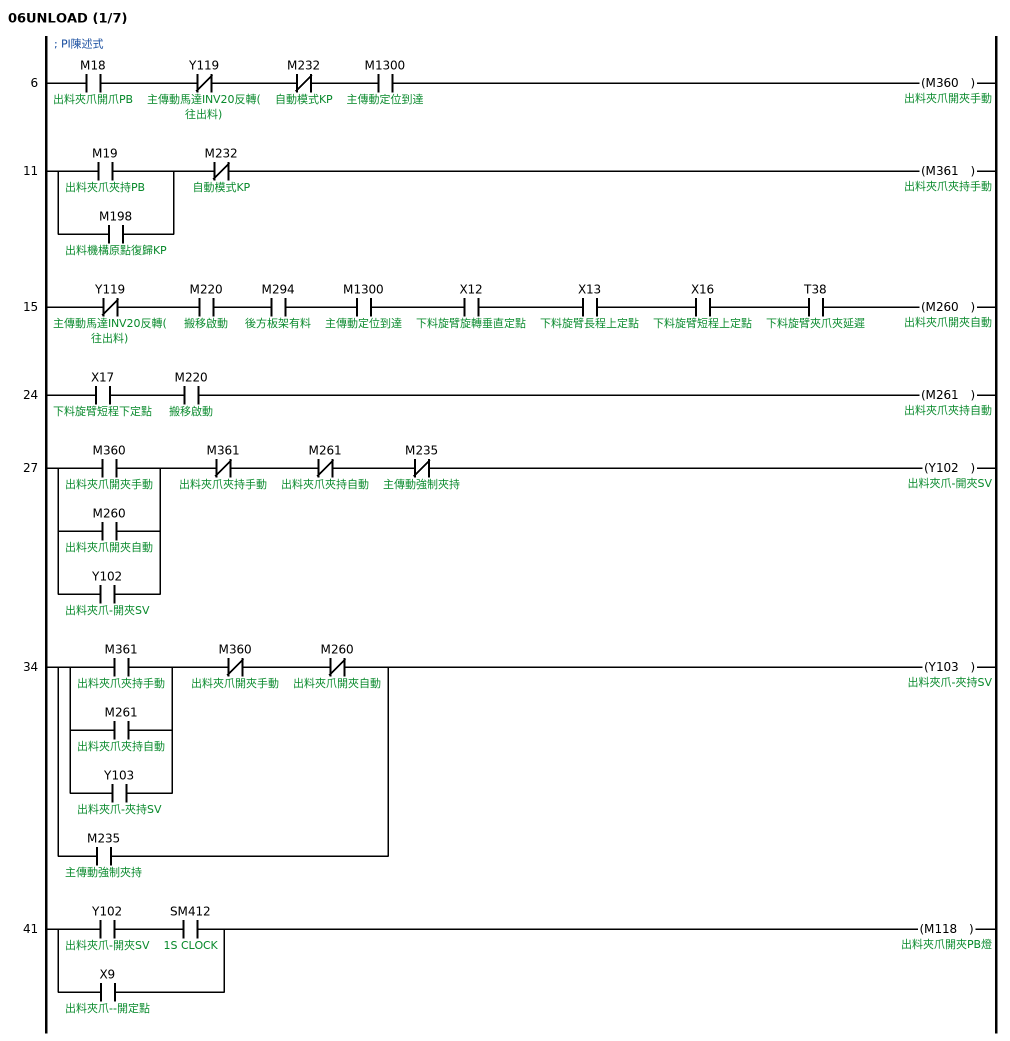
[picture p24: ladder of 06UNLOAD, rungs at steps 6 to 41]
; PI陳述式
6     LD      M18  ; 出料夾爪開爪PB
      ANI     Y119  ; 主傳動馬達INV20反轉(往出料)
      ANI     M232  ; 自動模式KP
      AND     M1300  ; 主傳動定位到達
      OUT     M360  ; 出料夾爪開夾手動
11    LD      M19  ; 出料夾爪夾持PB
      OR      M198  ; 出料機構原點復歸KP
      ANI     M232  ; 自動模式KP
      OUT     M361  ; 出料夾爪夾持手動
15    LDI     Y119  ; 主傳動馬達INV20反轉(往出料)
      AND     M220  ; 搬移啟動
      AND     M294  ; 後方板架有料
      AND     M1300  ; 主傳動定位到達
      AND     X12  ; 下料旋臂旋轉垂直定點
      AND     X13  ; 下料旋臂長程上定點
      AND     X16  ; 下料旋臂短程上定點
      AND     T38  ; 下料旋臂夾爪夾延遲
      OUT     M260  ; 出料夾爪開夾自動
24    LD      X17  ; 下料旋臂短程下定點
      AND     M220  ; 搬移啟動
      OUT     M261  ; 出料夾爪夾持自動
27    LD      M360  ; 出料夾爪開夾手動
      OR      M260  ; 出料夾爪開夾自動
      OR      Y102  ; 出料夾爪-開夾SV
      ANI     M361  ; 出料夾爪夾持手動
      ANI     M261  ; 出料夾爪夾持自動
      ANI     M235  ; 主傳動強制夾持
      OUT     Y102  ; 出料夾爪-開夾SV
34    LD      M361  ; 出料夾爪夾持手動
      OR      M261  ; 出料夾爪夾持自動
      OR      Y103  ; 出料夾爪-夾持SV
      ANI     M360  ; 出料夾爪開夾手動
      ANI     M260  ; 出料夾爪開夾自動
      OR      M235  ; 主傳動強制夾持
      OUT     Y103  ; 出料夾爪-夾持SV
41    LD      Y102  ; 出料夾爪-開夾SV
      AND     SM412  ; 1S CLOCK
      OR      X9  ; 出料夾爪--開定點
      OUT     M118  ; 出料夾爪開夾PB燈
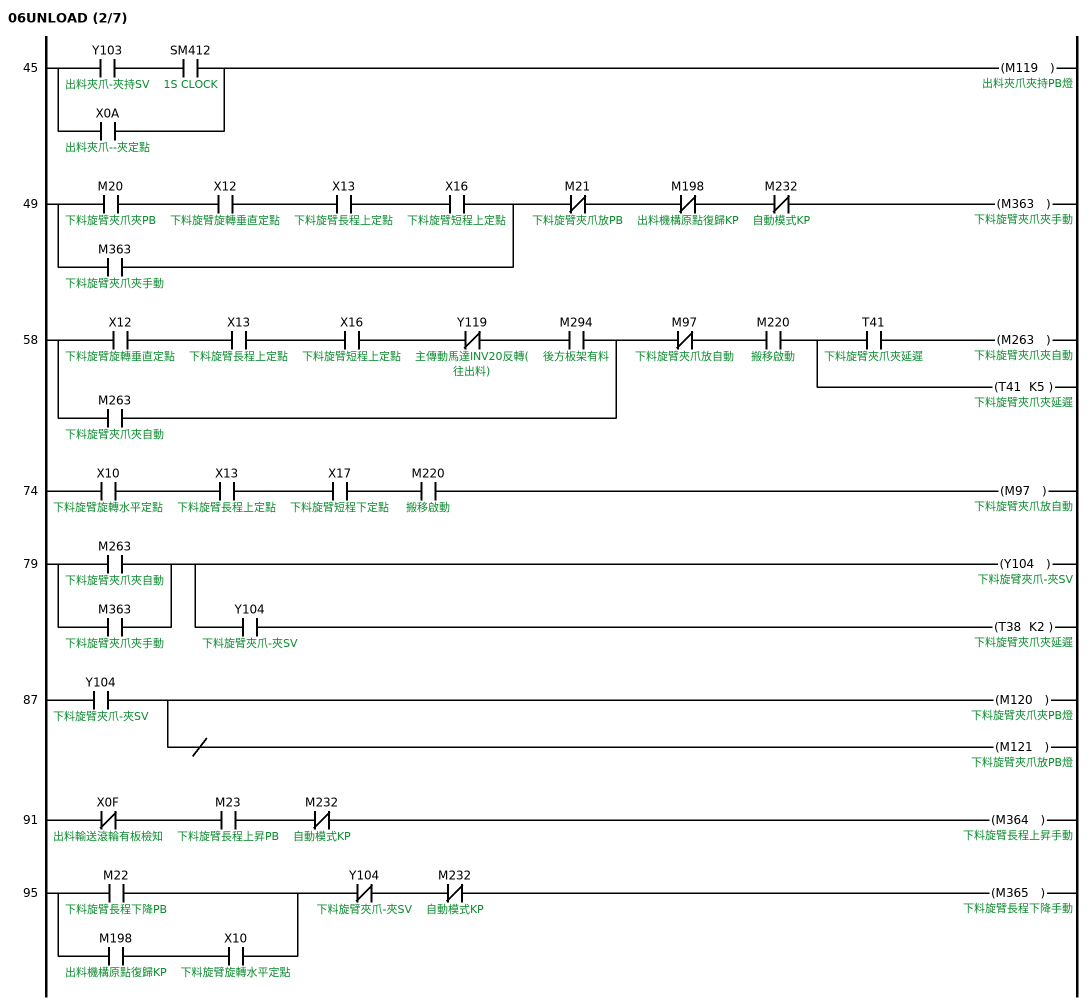
45    LD      Y103  ; 出料夾爪-夾持SV
      AND     SM412  ; 1S CLOCK
      OR      X0A  ; 出料夾爪--夾定點
      OUT     M119  ; 出料夾爪夾持PB燈
49    LD      M20  ; 下料旋臂夾爪夾PB
      AND     X12  ; 下料旋臂旋轉垂直定點
      AND     X13  ; 下料旋臂長程上定點
      AND     X16  ; 下料旋臂短程上定點
      OR      M363  ; 下料旋臂夾爪夾手動
      ANI     M21  ; 下料旋臂夾爪放PB
      ANI     M198  ; 出料機構原點復歸KP
      ANI     M232  ; 自動模式KP
      OUT     M363  ; 下料旋臂夾爪夾手動
58    LD      X12  ; 下料旋臂旋轉垂直定點
      AND     X13  ; 下料旋臂長程上定點
      AND     X16  ; 下料旋臂短程上定點
      ANI     Y119  ; 主傳動馬達INV20反轉(往出料)
      AND     M294  ; 後方板架有料
      OR      M263  ; 下料旋臂夾爪夾自動
      ANI     M97  ; 下料旋臂夾爪放自動
      AND     M220  ; 搬移啟動
      MPS
      AND     T41  ; 下料旋臂夾爪夾延遲
      OUT     M263  ; 下料旋臂夾爪夾自動
      MPP
      OUT     T41 K5  ; 下料旋臂夾爪夾延遲
74    LD      X10  ; 下料旋臂旋轉水平定點
      AND     X13  ; 下料旋臂長程上定點
      AND     X17  ; 下料旋臂短程下定點
      AND     M220  ; 搬移啟動
      OUT     M97  ; 下料旋臂夾爪放自動
79    LD      M263  ; 下料旋臂夾爪夾自動
      OR      M363  ; 下料旋臂夾爪夾手動
      OUT     Y104  ; 下料旋臂夾爪-夾SV
      AND     Y104  ; 下料旋臂夾爪-夾SV
      OUT     T38 K2  ; 下料旋臂夾爪夾延遲
87    LD      Y104  ; 下料旋臂夾爪-夾SV
      OUT     M120  ; 下料旋臂夾爪夾PB燈
      INV
      OUT     M121  ; 下料旋臂夾爪放PB燈
91    LDI     X0F  ; 出料輸送滾輪有板檢知
      AND     M23  ; 下料旋臂長程上昇PB
      ANI     M232  ; 自動模式KP
      OUT     M364  ; 下料旋臂長程上昇手動
95    LD      M22  ; 下料旋臂長程下降PB
      LD      M198  ; 出料機構原點復歸KP
      AND     X10  ; 下料旋臂旋轉水平定點
      ORB
      ANI     Y104  ; 下料旋臂夾爪-夾SV
      ANI     M232  ; 自動模式KP
      OUT     M365  ; 下料旋臂長程下降手動
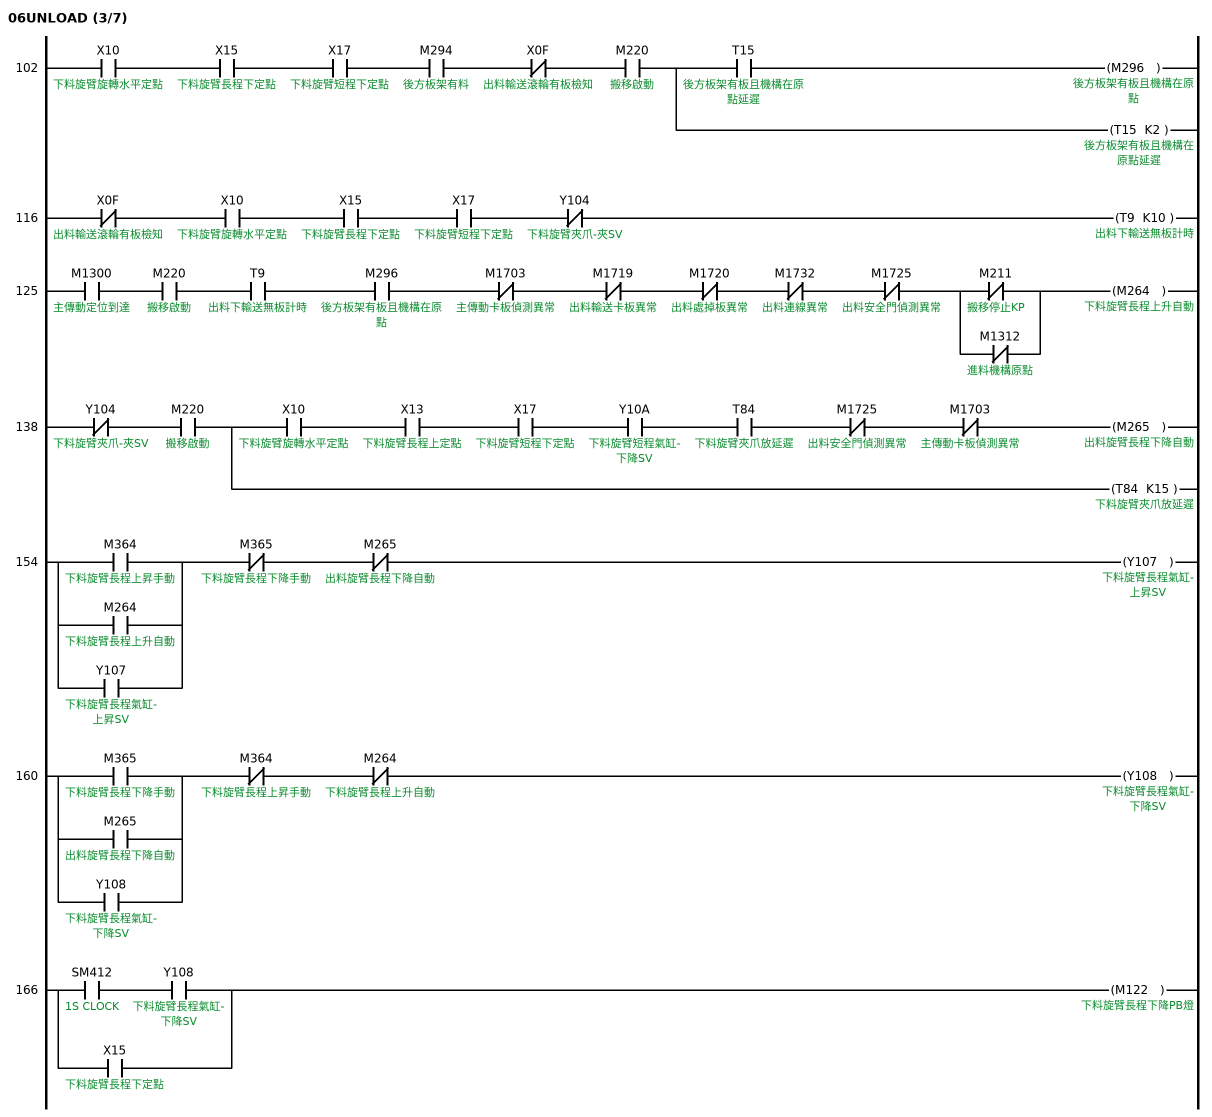
102   LD      X10  ; 下料旋臂旋轉水平定點
      AND     X15  ; 下料旋臂長程下定點
      AND     X17  ; 下料旋臂短程下定點
      AND     M294  ; 後方板架有料
      ANI     X0F  ; 出料輸送滾輪有板檢知
      AND     M220  ; 搬移啟動
      MPS
      AND     T15  ; 後方板架有板且機構在原點延遲
      OUT     M296  ; 後方板架有板且機構在原點
      MPP
      OUT     T15 K2  ; 後方板架有板且機構在原點延遲
116   LDI     X0F  ; 出料輸送滾輪有板檢知
      AND     X10  ; 下料旋臂旋轉水平定點
      AND     X15  ; 下料旋臂長程下定點
      AND     X17  ; 下料旋臂短程下定點
      ANI     Y104  ; 下料旋臂夾爪-夾SV
      OUT     T9 K10  ; 出料下輸送無板計時
125   LD      M1300  ; 主傳動定位到達
      AND     M220  ; 搬移啟動
      AND     T9  ; 出料下輸送無板計時
      AND     M296  ; 後方板架有板且機構在原點
      ANI     M1703  ; 主傳動卡板偵測異常
      ANI     M1719  ; 出料輸送卡板異常
      ANI     M1720  ; 出料處掉板異常
      ANI     M1732  ; 出料連線異常
      ANI     M1725  ; 出料安全門偵測異常
      LDI     M211  ; 搬移停止KP
      ORI     M1312  ; 進料機構原點
      ANB
      OUT     M264  ; 下料旋臂長程上升自動
138   LDI     Y104  ; 下料旋臂夾爪-夾SV
      AND     M220  ; 搬移啟動
      MPS
      AND     X10  ; 下料旋臂旋轉水平定點
      AND     X13  ; 下料旋臂長程上定點
      AND     X17  ; 下料旋臂短程下定點
      AND     Y10A  ; 下料旋臂短程氣缸-下降SV
      AND     T84  ; 下料旋臂夾爪放延遲
      ANI     M1725  ; 出料安全門偵測異常
      ANI     M1703  ; 主傳動卡板偵測異常
      OUT     M265  ; 出料旋臂長程下降自動
      MPP
      OUT     T84 K15  ; 下料旋臂夾爪放延遲
154   LD      M364  ; 下料旋臂長程上昇手動
      OR      M264  ; 下料旋臂長程上升自動
      OR      Y107  ; 下料旋臂長程氣缸-上昇SV
      ANI     M365  ; 下料旋臂長程下降手動
      ANI     M265  ; 出料旋臂長程下降自動
      OUT     Y107  ; 下料旋臂長程氣缸-上昇SV
160   LD      M365  ; 下料旋臂長程下降手動
      OR      M265  ; 出料旋臂長程下降自動
      OR      Y108  ; 下料旋臂長程氣缸-下降SV
      ANI     M364  ; 下料旋臂長程上昇手動
      ANI     M264  ; 下料旋臂長程上升自動
      OUT     Y108  ; 下料旋臂長程氣缸-下降SV
166   LD      SM412  ; 1S CLOCK
      AND     Y108  ; 下料旋臂長程氣缸-下降SV
      OR      X15  ; 下料旋臂長程下定點
      OUT     M122  ; 下料旋臂長程下降PB燈
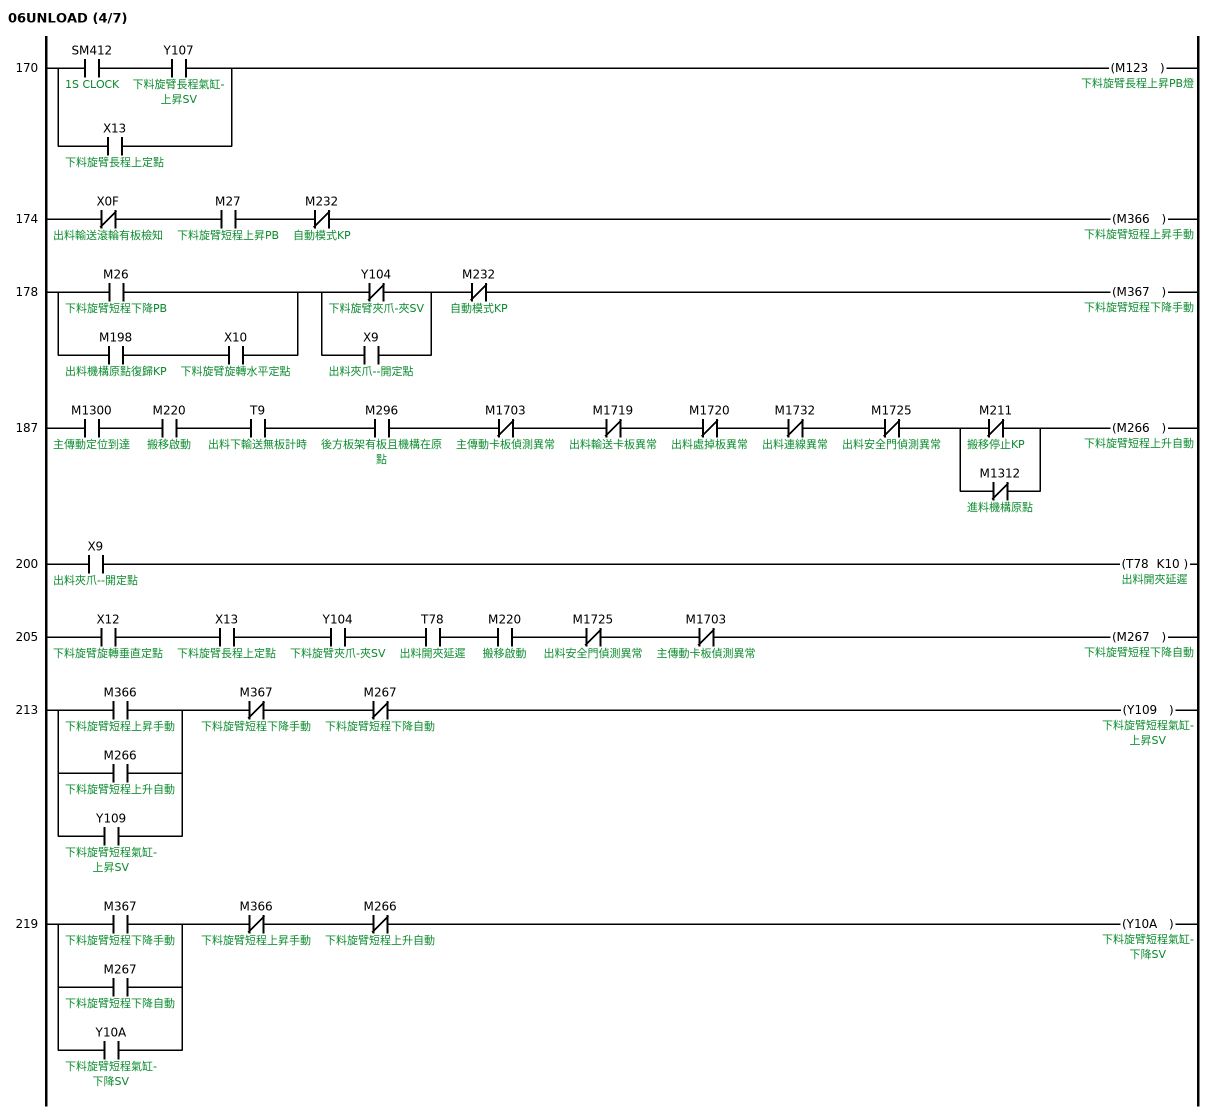
170   LD      SM412  ; 1S CLOCK
      AND     Y107  ; 下料旋臂長程氣缸-上昇SV
      OR      X13  ; 下料旋臂長程上定點
      OUT     M123  ; 下料旋臂長程上昇PB燈
174   LDI     X0F  ; 出料輸送滾輪有板檢知
      AND     M27  ; 下料旋臂短程上昇PB
      ANI     M232  ; 自動模式KP
      OUT     M366  ; 下料旋臂短程上昇手動
178   LD      M26  ; 下料旋臂短程下降PB
      LD      M198  ; 出料機構原點復歸KP
      AND     X10  ; 下料旋臂旋轉水平定點
      ORB
      LDI     Y104  ; 下料旋臂夾爪-夾SV
      OR      X9  ; 出料夾爪--開定點
      ANB
      ANI     M232  ; 自動模式KP
      OUT     M367  ; 下料旋臂短程下降手動
187   LD      M1300  ; 主傳動定位到達
      AND     M220  ; 搬移啟動
      AND     T9  ; 出料下輸送無板計時
      AND     M296  ; 後方板架有板且機構在原點
      ANI     M1703  ; 主傳動卡板偵測異常
      ANI     M1719  ; 出料輸送卡板異常
      ANI     M1720  ; 出料處掉板異常
      ANI     M1732  ; 出料連線異常
      ANI     M1725  ; 出料安全門偵測異常
      LDI     M211  ; 搬移停止KP
      ORI     M1312  ; 進料機構原點
      ANB
      OUT     M266  ; 下料旋臂短程上升自動
200   LD      X9  ; 出料夾爪--開定點
      OUT     T78 K10  ; 出料開夾延遲
205   LD      X12  ; 下料旋臂旋轉垂直定點
      AND     X13  ; 下料旋臂長程上定點
      AND     Y104  ; 下料旋臂夾爪-夾SV
      AND     T78  ; 出料開夾延遲
      AND     M220  ; 搬移啟動
      ANI     M1725  ; 出料安全門偵測異常
      ANI     M1703  ; 主傳動卡板偵測異常
      OUT     M267  ; 下料旋臂短程下降自動
213   LD      M366  ; 下料旋臂短程上昇手動
      OR      M266  ; 下料旋臂短程上升自動
      OR      Y109  ; 下料旋臂短程氣缸-上昇SV
      ANI     M367  ; 下料旋臂短程下降手動
      ANI     M267  ; 下料旋臂短程下降自動
      OUT     Y109  ; 下料旋臂短程氣缸-上昇SV
219   LD      M367  ; 下料旋臂短程下降手動
      OR      M267  ; 下料旋臂短程下降自動
      OR      Y10A  ; 下料旋臂短程氣缸-下降SV
      ANI     M366  ; 下料旋臂短程上昇手動
      ANI     M266  ; 下料旋臂短程上升自動
      OUT     Y10A  ; 下料旋臂短程氣缸-下降SV
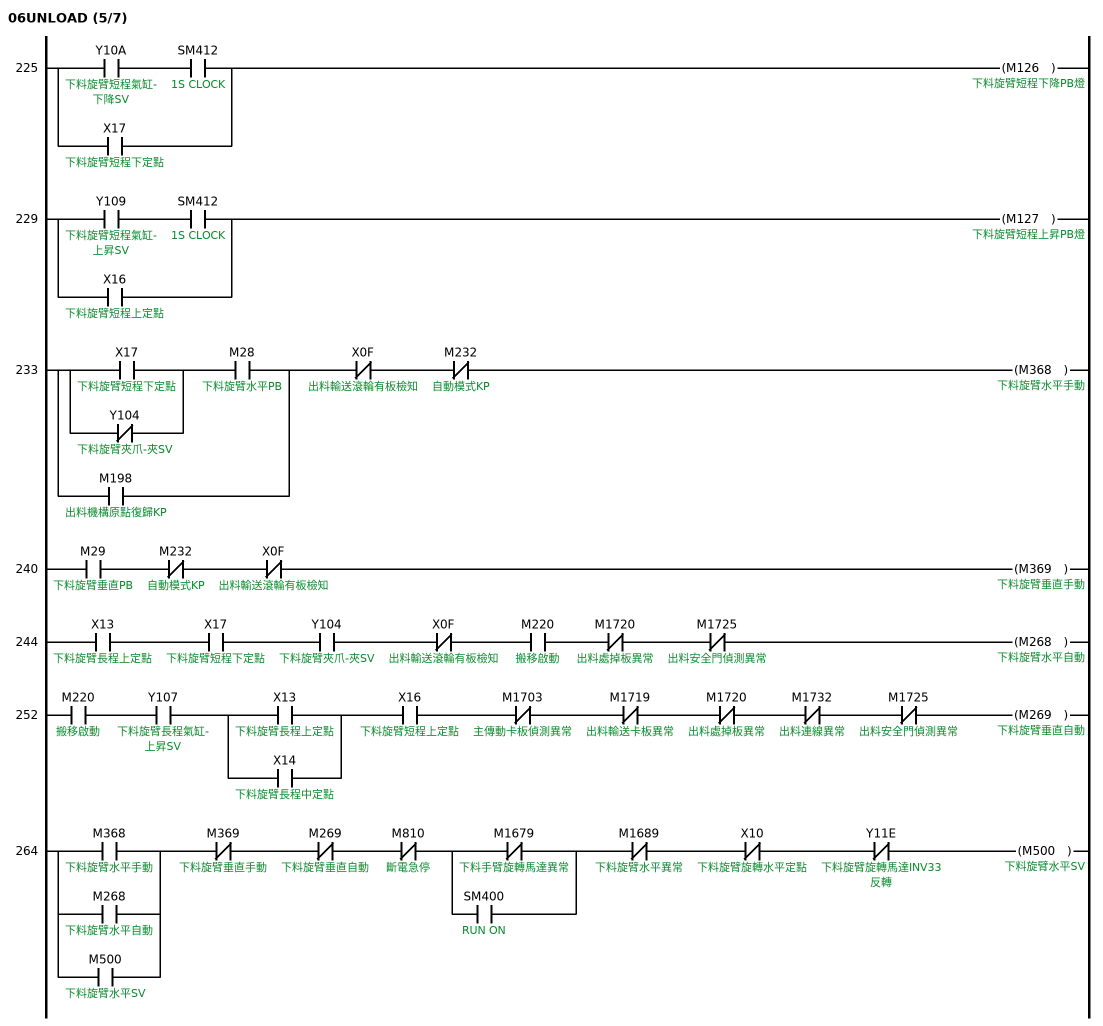
225   LD      Y10A  ; 下料旋臂短程氣缸-下降SV
      AND     SM412  ; 1S CLOCK
      OR      X17  ; 下料旋臂短程下定點
      OUT     M126  ; 下料旋臂短程下降PB燈
229   LD      Y109  ; 下料旋臂短程氣缸-上昇SV
      AND     SM412  ; 1S CLOCK
      OR      X16  ; 下料旋臂短程上定點
      OUT     M127  ; 下料旋臂短程上昇PB燈
233   LD      X17  ; 下料旋臂短程下定點
      ORI     Y104  ; 下料旋臂夾爪-夾SV
      AND     M28  ; 下料旋臂水平PB
      OR      M198  ; 出料機構原點復歸KP
      ANI     X0F  ; 出料輸送滾輪有板檢知
      ANI     M232  ; 自動模式KP
      OUT     M368  ; 下料旋臂水平手動
240   LD      M29  ; 下料旋臂垂直PB
      ANI     M232  ; 自動模式KP
      ANI     X0F  ; 出料輸送滾輪有板檢知
      OUT     M369  ; 下料旋臂垂直手動
244   LD      X13  ; 下料旋臂長程上定點
      AND     X17  ; 下料旋臂短程下定點
      AND     Y104  ; 下料旋臂夾爪-夾SV
      ANI     X0F  ; 出料輸送滾輪有板檢知
      AND     M220  ; 搬移啟動
      ANI     M1720  ; 出料處掉板異常
      ANI     M1725  ; 出料安全門偵測異常
      OUT     M268  ; 下料旋臂水平自動
252   LD      M220  ; 搬移啟動
      AND     Y107  ; 下料旋臂長程氣缸-上昇SV
      LD      X13  ; 下料旋臂長程上定點
      OR      X14  ; 下料旋臂長程中定點
      ANB
      AND     X16  ; 下料旋臂短程上定點
      ANI     M1703  ; 主傳動卡板偵測異常
      ANI     M1719  ; 出料輸送卡板異常
      ANI     M1720  ; 出料處掉板異常
      ANI     M1732  ; 出料連線異常
      ANI     M1725  ; 出料安全門偵測異常
      OUT     M269  ; 下料旋臂垂直自動
264   LD      M368  ; 下料旋臂水平手動
      OR      M268  ; 下料旋臂水平自動
      OR      M500  ; 下料旋臂水平SV
      ANI     M369  ; 下料旋臂垂直手動
      ANI     M269  ; 下料旋臂垂直自動
      ANI     M810  ; 斷電急停
      LDI     M1679  ; 下料手臂旋轉馬達異常
      OR      SM400  ; RUN ON
      ANB
      ANI     M1689  ; 下料旋臂水平異常
      ANI     X10  ; 下料旋臂旋轉水平定點
      ANI     Y11E  ; 下料旋臂旋轉馬達INV33反轉
      OUT     M500  ; 下料旋臂水平SV
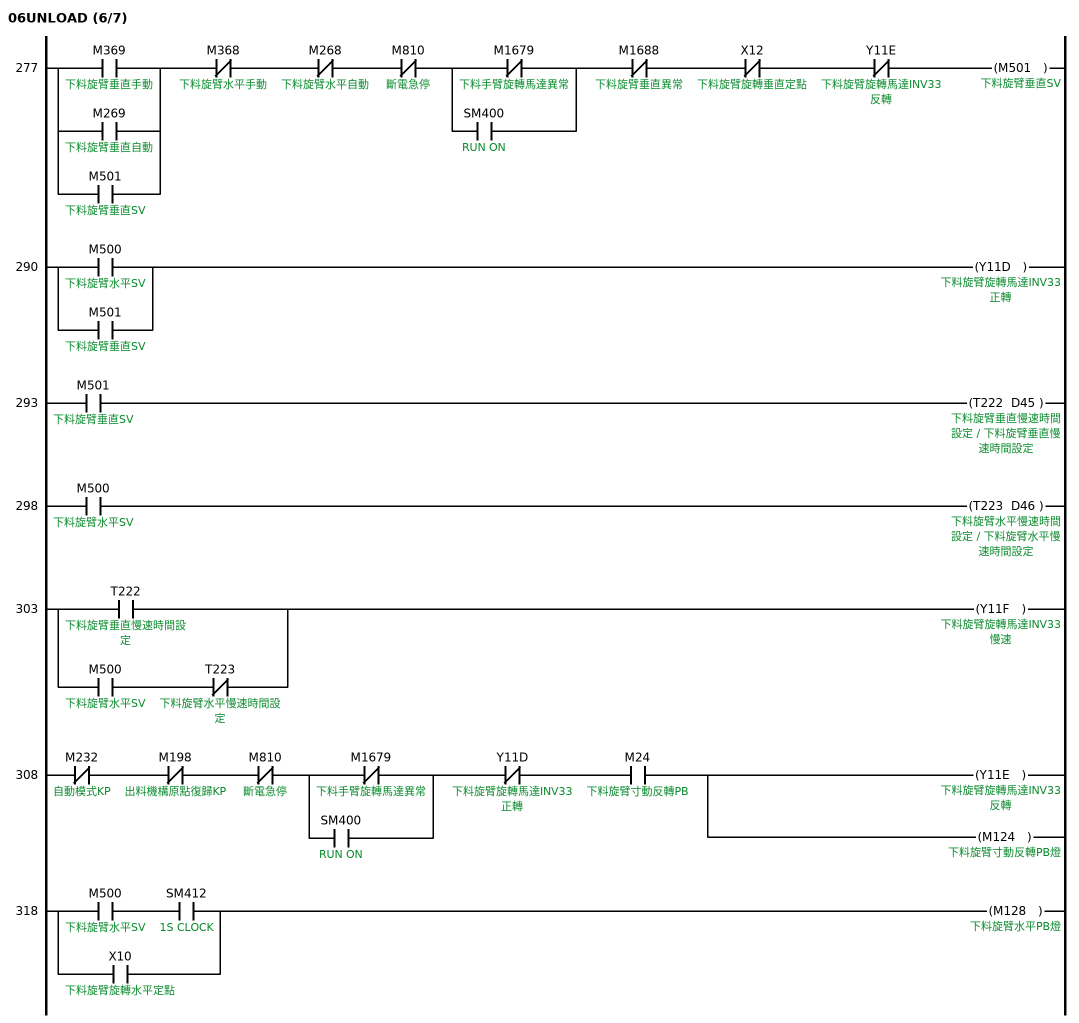
277   LD      M369  ; 下料旋臂垂直手動
      OR      M269  ; 下料旋臂垂直自動
      OR      M501  ; 下料旋臂垂直SV
      ANI     M368  ; 下料旋臂水平手動
      ANI     M268  ; 下料旋臂水平自動
      ANI     M810  ; 斷電急停
      LDI     M1679  ; 下料手臂旋轉馬達異常
      OR      SM400  ; RUN ON
      ANB
      ANI     M1688  ; 下料旋臂垂直異常
      ANI     X12  ; 下料旋臂旋轉垂直定點
      ANI     Y11E  ; 下料旋臂旋轉馬達INV33反轉
      OUT     M501  ; 下料旋臂垂直SV
290   LD      M500  ; 下料旋臂水平SV
      OR      M501  ; 下料旋臂垂直SV
      OUT     Y11D  ; 下料旋臂旋轉馬達INV33正轉
293   LD      M501  ; 下料旋臂垂直SV
      OUT     T222 D45  ; 下料旋臂垂直慢速時間設定 / 下料旋臂垂直慢速時間設定
298   LD      M500  ; 下料旋臂水平SV
      OUT     T223 D46  ; 下料旋臂水平慢速時間設定 / 下料旋臂水平慢速時間設定
303   LD      T222  ; 下料旋臂垂直慢速時間設定
      LD      M500  ; 下料旋臂水平SV
      ANI     T223  ; 下料旋臂水平慢速時間設定
      ORB
      OUT     Y11F  ; 下料旋臂旋轉馬達INV33慢速
308   LDI     M232  ; 自動模式KP
      ANI     M198  ; 出料機構原點復歸KP
      ANI     M810  ; 斷電急停
      LDI     M1679  ; 下料手臂旋轉馬達異常
      OR      SM400  ; RUN ON
      ANB
      ANI     Y11D  ; 下料旋臂旋轉馬達INV33正轉
      AND     M24  ; 下料旋臂寸動反轉PB
      OUT     Y11E  ; 下料旋臂旋轉馬達INV33反轉
      OUT     M124  ; 下料旋臂寸動反轉PB燈
318   LD      M500  ; 下料旋臂水平SV
      AND     SM412  ; 1S CLOCK
      OR      X10  ; 下料旋臂旋轉水平定點
      OUT     M128  ; 下料旋臂水平PB燈
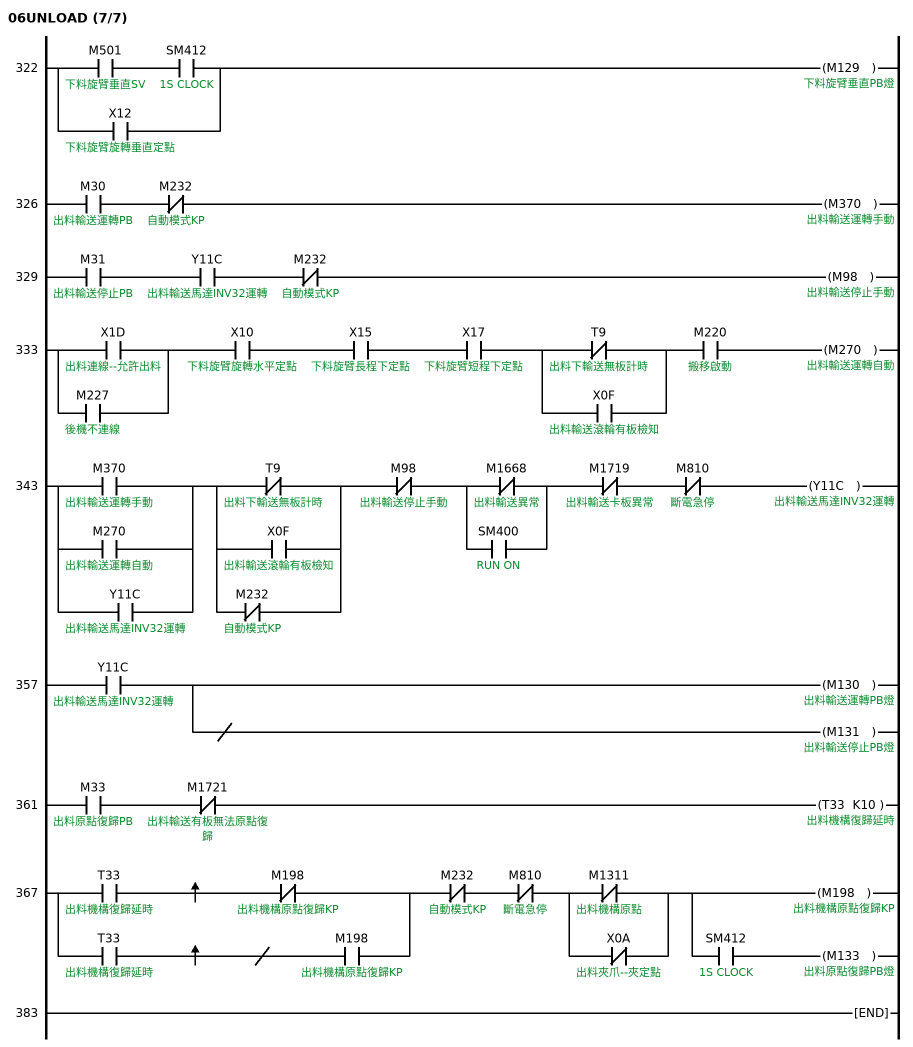
322   LD      M501  ; 下料旋臂垂直SV
      AND     SM412  ; 1S CLOCK
      OR      X12  ; 下料旋臂旋轉垂直定點
      OUT     M129  ; 下料旋臂垂直PB燈
326   LD      M30  ; 出料輸送運轉PB
      ANI     M232  ; 自動模式KP
      OUT     M370  ; 出料輸送運轉手動
329   LD      M31  ; 出料輸送停止PB
      AND     Y11C  ; 出料輸送馬達INV32運轉
      ANI     M232  ; 自動模式KP
      OUT     M98  ; 出料輸送停止手動
333   LD      X1D  ; 出料連線--允許出料
      OR      M227  ; 後機不連線
      AND     X10  ; 下料旋臂旋轉水平定點
      AND     X15  ; 下料旋臂長程下定點
      AND     X17  ; 下料旋臂短程下定點
      LDI     T9  ; 出料下輸送無板計時
      OR      X0F  ; 出料輸送滾輪有板檢知
      ANB
      AND     M220  ; 搬移啟動
      OUT     M270  ; 出料輸送運轉自動
343   LD      M370  ; 出料輸送運轉手動
      OR      M270  ; 出料輸送運轉自動
      OR      Y11C  ; 出料輸送馬達INV32運轉
      LDI     T9  ; 出料下輸送無板計時
      OR      X0F  ; 出料輸送滾輪有板檢知
      ORI     M232  ; 自動模式KP
      ANB
      ANI     M98  ; 出料輸送停止手動
      LDI     M1668  ; 出料輸送異常
      OR      SM400  ; RUN ON
      ANB
      ANI     M1719  ; 出料輸送卡板異常
      ANI     M810  ; 斷電急停
      OUT     Y11C  ; 出料輸送馬達INV32運轉
357   LD      Y11C  ; 出料輸送馬達INV32運轉
      OUT     M130  ; 出料輸送運轉PB燈
      INV
      OUT     M131  ; 出料輸送停止PB燈
361   LD      M33  ; 出料原點復歸PB
      ANI     M1721  ; 出料輸送有板無法原點復歸
      OUT     T33 K10  ; 出料機構復歸延時
367   LD      T33  ; 出料機構復歸延時
      MEP
      ANI     M198  ; 出料機構原點復歸KP
      LD      T33  ; 出料機構復歸延時
      MEP
      INV
      AND     M198  ; 出料機構原點復歸KP
      ORB
      ANI     M232  ; 自動模式KP
      ANI     M810  ; 斷電急停
      LDI     M1311  ; 出料機構原點
      ORI     X0A  ; 出料夾爪--夾定點
      ANB
      OUT     M198  ; 出料機構原點復歸KP
      AND     SM412  ; 1S CLOCK
      OUT     M133  ; 出料原點復歸PB燈
383   END
END_PROGRAM

PROGRAM 07UNMOVE
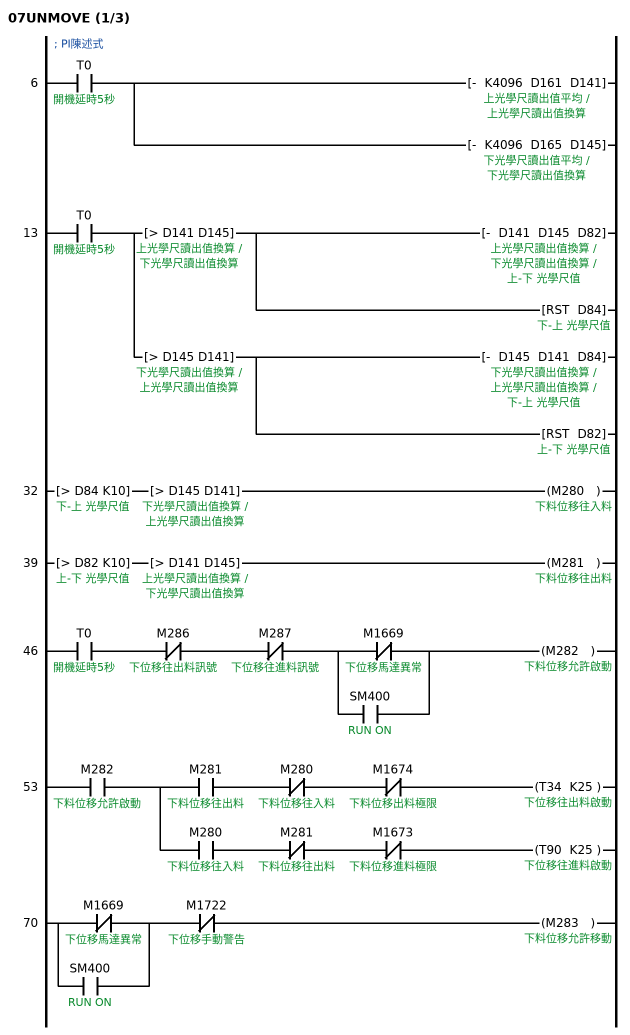
; PI陳述式
6     LD      T0  ; 開機延時5秒
      -       K4096 D161 D141  ; 上光學尺讀出值平均 / 上光學尺讀出值換算
      -       K4096 D165 D145  ; 下光學尺讀出值平均 / 下光學尺讀出值換算
13    LD      T0  ; 開機延時5秒
      MPS
      AND>    D141 D145  ; 上光學尺讀出值換算 / 下光學尺讀出值換算
      -       D141 D145 D82  ; 上-下 光學尺值
      RST     D84  ; 下-上 光學尺值
      MPP
      AND>    D145 D141  ; 下光學尺讀出值換算 / 上光學尺讀出值換算
      -       D145 D141 D84
      RST     D82  ; 上-下 光學尺值
32    LD>     D84 K10  ; 下-上 光學尺值
      AND>    D145 D141  ; 下光學尺讀出值換算 / 上光學尺讀出值換算
      OUT     M280  ; 下料位移往入料
39    LD>     D82 K10  ; 上-下 光學尺值
      AND>    D141 D145  ; 上光學尺讀出值換算 / 下光學尺讀出值換算
      OUT     M281  ; 下料位移往出料
46    LD      T0  ; 開機延時5秒
      ANI     M286  ; 下位移往出料訊號
      ANI     M287  ; 下位移往進料訊號
      LDI     M1669  ; 下位移馬達異常
      OR      SM400  ; RUN ON
      ANB
      OUT     M282  ; 下料位移允許啟動
53    LD      M282  ; 下料位移允許啟動
      MPS
      AND     M281  ; 下料位移往出料
      ANI     M280  ; 下料位移往入料
      ANI     M1674  ; 下料位移出料極限
      OUT     T34 K25  ; 下位移往出料啟動
      MPP
      AND     M280  ; 下料位移往入料
      ANI     M281  ; 下料位移往出料
      ANI     M1673  ; 下料位移進料極限
      OUT     T90 K25  ; 下位移往進料啟動
70    LDI     M1669  ; 下位移馬達異常
      OR      SM400  ; RUN ON
      ANI     M1722  ; 下位移手動警告
      OUT     M283  ; 下料位移允許移動
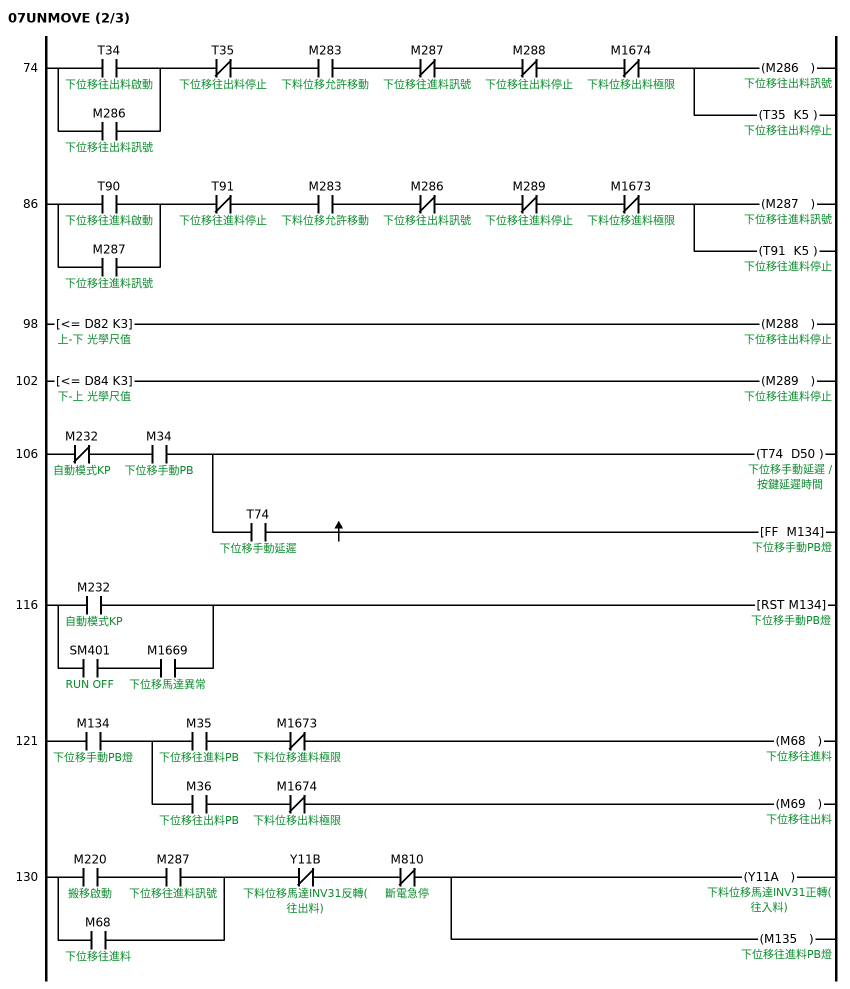
74    LD      T34  ; 下位移往出料啟動
      OR      M286  ; 下位移往出料訊號
      ANI     T35  ; 下位移往出料停止
      AND     M283  ; 下料位移允許移動
      ANI     M287  ; 下位移往進料訊號
      ANI     M288  ; 下位移往出料停止
      ANI     M1674  ; 下料位移出料極限
      OUT     M286  ; 下位移往出料訊號
      OUT     T35 K5  ; 下位移往出料停止
86    LD      T90  ; 下位移往進料啟動
      OR      M287  ; 下位移往進料訊號
      ANI     T91  ; 下位移往進料停止
      AND     M283  ; 下料位移允許移動
      ANI     M286  ; 下位移往出料訊號
      ANI     M289  ; 下位移往進料停止
      ANI     M1673  ; 下料位移進料極限
      OUT     M287  ; 下位移往進料訊號
      OUT     T91 K5  ; 下位移往進料停止
98    LD<=    D82 K3  ; 上-下 光學尺值
      OUT     M288  ; 下位移往出料停止
102   LD<=    D84 K3  ; 下-上 光學尺值
      OUT     M289  ; 下位移往進料停止
106   LDI     M232  ; 自動模式KP
      AND     M34  ; 下位移手動PB
      OUT     T74 D50  ; 下位移手動延遲 / 按鍵延遲時間
      AND     T74  ; 下位移手動延遲
      MEP
      FF      M134  ; 下位移手動PB燈
116   LD      M232  ; 自動模式KP
      LD      SM401  ; RUN OFF
      AND     M1669  ; 下位移馬達異常
      ORB
      RST     M134  ; 下位移手動PB燈
121   LD      M134  ; 下位移手動PB燈
      MPS
      AND     M35  ; 下位移往進料PB
      ANI     M1673  ; 下料位移進料極限
      OUT     M68  ; 下位移往進料
      MPP
      AND     M36  ; 下位移往出料PB
      ANI     M1674  ; 下料位移出料極限
      OUT     M69  ; 下位移往出料
130   LD      M220  ; 搬移啟動
      AND     M287  ; 下位移往進料訊號
      OR      M68  ; 下位移往進料
      ANI     Y11B  ; 下料位移馬達INV31反轉(往出料)
      ANI     M810  ; 斷電急停
      OUT     Y11A  ; 下料位移馬達INV31正轉(往入料)
      OUT     M135  ; 下位移往進料PB燈
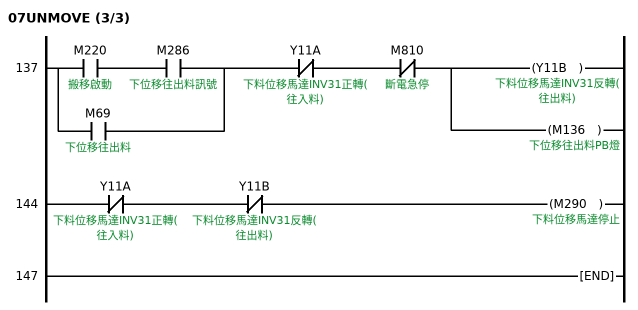
137   LD      M220  ; 搬移啟動
      AND     M286  ; 下位移往出料訊號
      OR      M69  ; 下位移往出料
      ANI     Y11A  ; 下料位移馬達INV31正轉(往入料)
      ANI     M810  ; 斷電急停
      OUT     Y11B  ; 下料位移馬達INV31反轉(往出料)
      OUT     M136  ; 下位移往出料PB燈
144   LDI     Y11A  ; 下料位移馬達INV31正轉(往入料)
      ANI     Y11B  ; 下料位移馬達INV31反轉(往出料)
      OUT     M290  ; 下料位移馬達停止
147   END
END_PROGRAM

PROGRAM 08HEATER
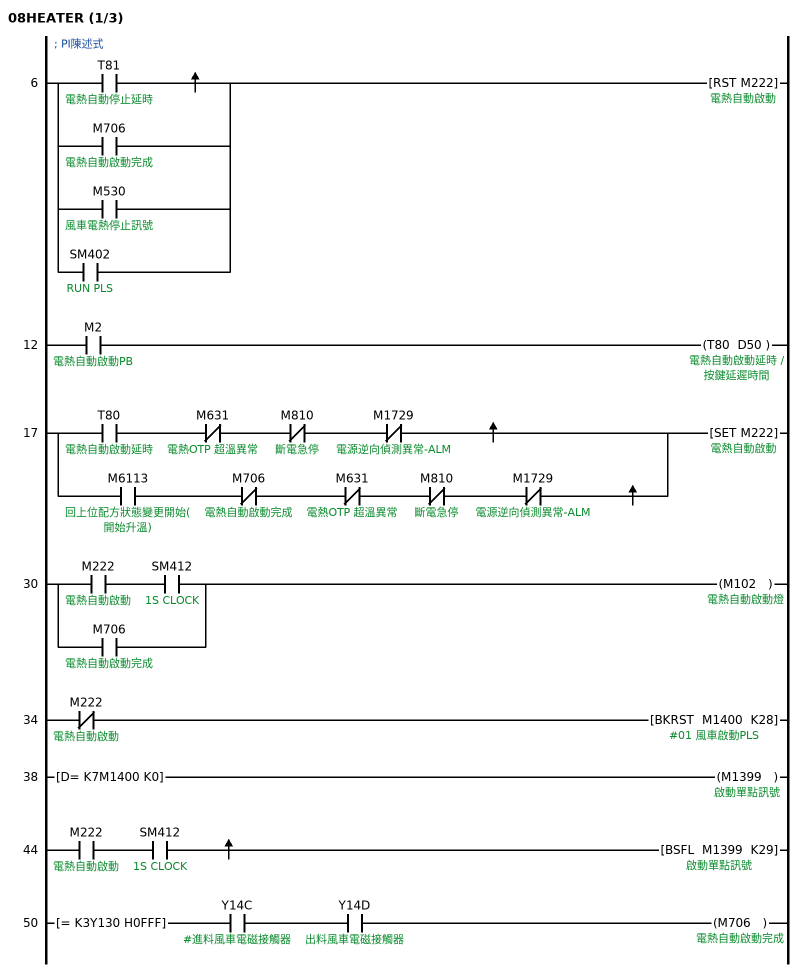
; PI陳述式
6     LD      T81  ; 電熱自動停止延時
      MEP
      OR      M706  ; 電熱自動啟動完成
      OR      M530  ; 風車電熱停止訊號
      OR      SM402  ; RUN PLS
      RST     M222  ; 電熱自動啟動
12    LD      M2  ; 電熱自動啟動PB
      OUT     T80 D50  ; 電熱自動啟動延時 / 按鍵延遲時間
17    LD      T80  ; 電熱自動啟動延時
      ANI     M631  ; 電熱OTP 超溫異常
      ANI     M810  ; 斷電急停
      ANI     M1729  ; 電源逆向偵測異常-ALM
      MEP
      LD      M6113  ; 回上位配方狀態變更開始(開始升溫)
      ANI     M706  ; 電熱自動啟動完成
      ANI     M631  ; 電熱OTP 超溫異常
      ANI     M810  ; 斷電急停
      ANI     M1729  ; 電源逆向偵測異常-ALM
      MEP
      ORB
      SET     M222  ; 電熱自動啟動
30    LD      M222  ; 電熱自動啟動
      AND     SM412  ; 1S CLOCK
      OR      M706  ; 電熱自動啟動完成
      OUT     M102  ; 電熱自動啟動燈
34    LDI     M222  ; 電熱自動啟動
      BKRST   M1400 K28  ; #01 風車啟動PLS
38    LDD=    K7M1400 K0  ; #01 風車啟動PLS
      OUT     M1399  ; 啟動單點訊號
44    LD      M222  ; 電熱自動啟動
      AND     SM412  ; 1S CLOCK
      MEP
      BSFL    M1399 K29
50    LD=     K3Y130 H0FFF  ; NO.01   加熱器電磁接觸器
      AND     Y14C  ; #進料風車電磁接觸器
      AND     Y14D  ; 出料風車電磁接觸器
      OUT     M706  ; 電熱自動啟動完成
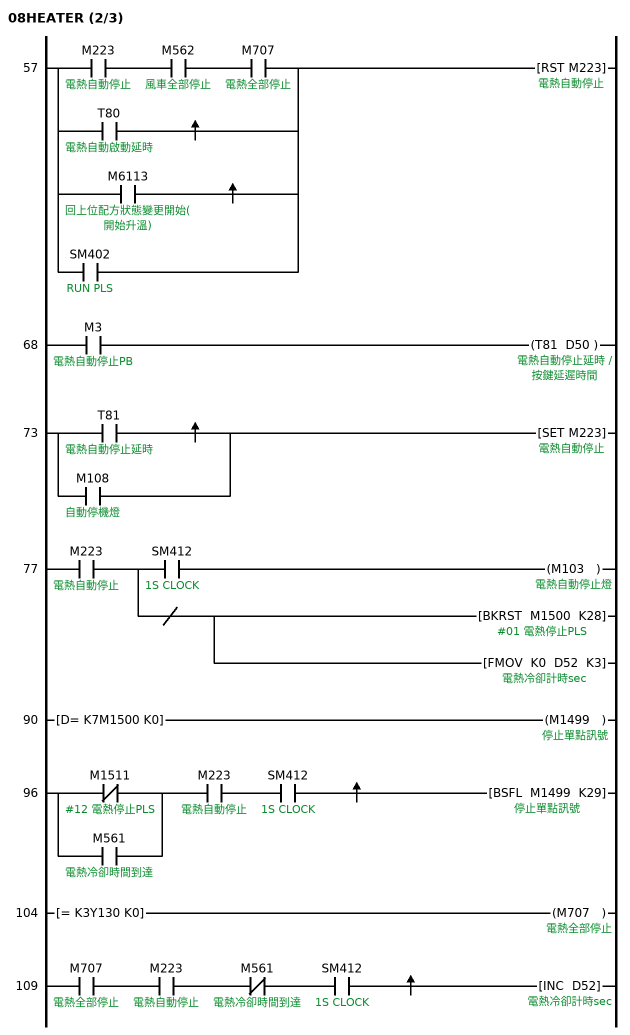
57    LD      M223  ; 電熱自動停止
      AND     M562  ; 風車全部停止
      AND     M707  ; 電熱全部停止
      LD      T80  ; 電熱自動啟動延時
      MEP
      ORB
      LD      M6113  ; 回上位配方狀態變更開始(開始升溫)
      MEP
      ORB
      OR      SM402  ; RUN PLS
      RST     M223  ; 電熱自動停止
68    LD      M3  ; 電熱自動停止PB
      OUT     T81 D50  ; 電熱自動停止延時 / 按鍵延遲時間
73    LD      T81  ; 電熱自動停止延時
      MEP
      OR      M108  ; 自動停機燈
      SET     M223  ; 電熱自動停止
77    LD      M223  ; 電熱自動停止
      MPS
      AND     SM412  ; 1S CLOCK
      OUT     M103  ; 電熱自動停止燈
      MPP
      INV
      BKRST   M1500 K28  ; #01 電熱停止PLS
      FMOV    K0 D52 K3  ; 電熱冷卻計時sec
90    LDD=    K7M1500 K0  ; #01 電熱停止PLS
      OUT     M1499  ; 停止單點訊號
96    LDI     M1511  ; #12 電熱停止PLS
      OR      M561  ; 電熱冷卻時間到達
      AND     M223  ; 電熱自動停止
      AND     SM412  ; 1S CLOCK
      MEP
      BSFL    M1499 K29
104   LD=     K3Y130 K0  ; NO.01   加熱器電磁接觸器
      OUT     M707  ; 電熱全部停止
109   LD      M707  ; 電熱全部停止
      AND     M223  ; 電熱自動停止
      ANI     M561  ; 電熱冷卻時間到達
      AND     SM412  ; 1S CLOCK
      MEP
      INC     D52
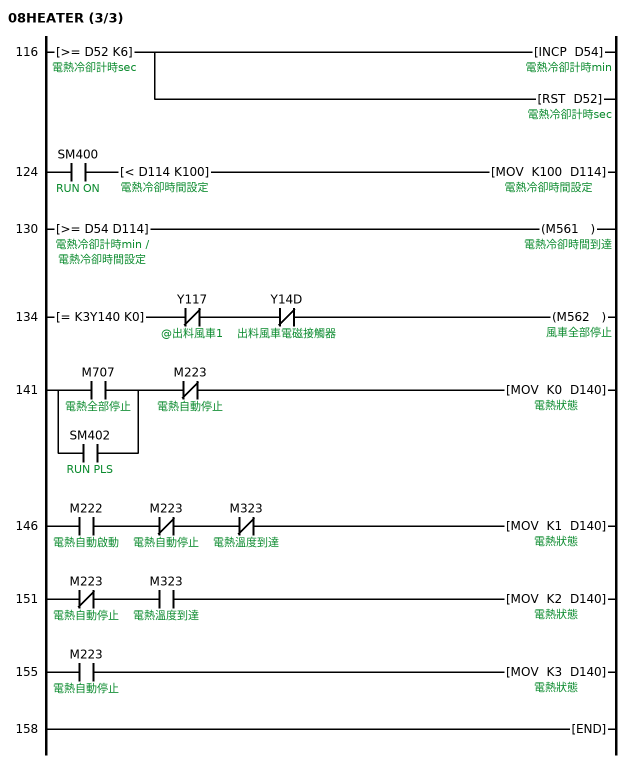
116   LD>=    D52 K6  ; 電熱冷卻計時sec
      INCP    D54  ; 電熱冷卻計時min
      RST     D52  ; 電熱冷卻計時sec
124   LD      SM400  ; RUN ON
      AND<    D114 K100  ; 電熱冷卻時間設定
      MOV     K100 D114
130   LD>=    D54 D114  ; 電熱冷卻計時min / 電熱冷卻時間設定
      OUT     M561  ; 電熱冷卻時間到達
134   LD=     K3Y140 K0  ; NO.01   風車電磁接觸器
      ANI     Y117  ; @出料風車1
      ANI     Y14D  ; 出料風車電磁接觸器
      OUT     M562  ; 風車全部停止
141   LD      M707  ; 電熱全部停止
      OR      SM402  ; RUN PLS
      ANI     M223  ; 電熱自動停止
      MOV     K0 D140  ; 電熱狀態
146   LD      M222  ; 電熱自動啟動
      ANI     M223  ; 電熱自動停止
      ANI     M323  ; 電熱溫度到達
      MOV     K1 D140
151   LDI     M223  ; 電熱自動停止
      AND     M323  ; 電熱溫度到達
      MOV     K2 D140
155   LD      M223  ; 電熱自動停止
      MOV     K3 D140
158   END
END_PROGRAM

PROGRAM 09BLOWER
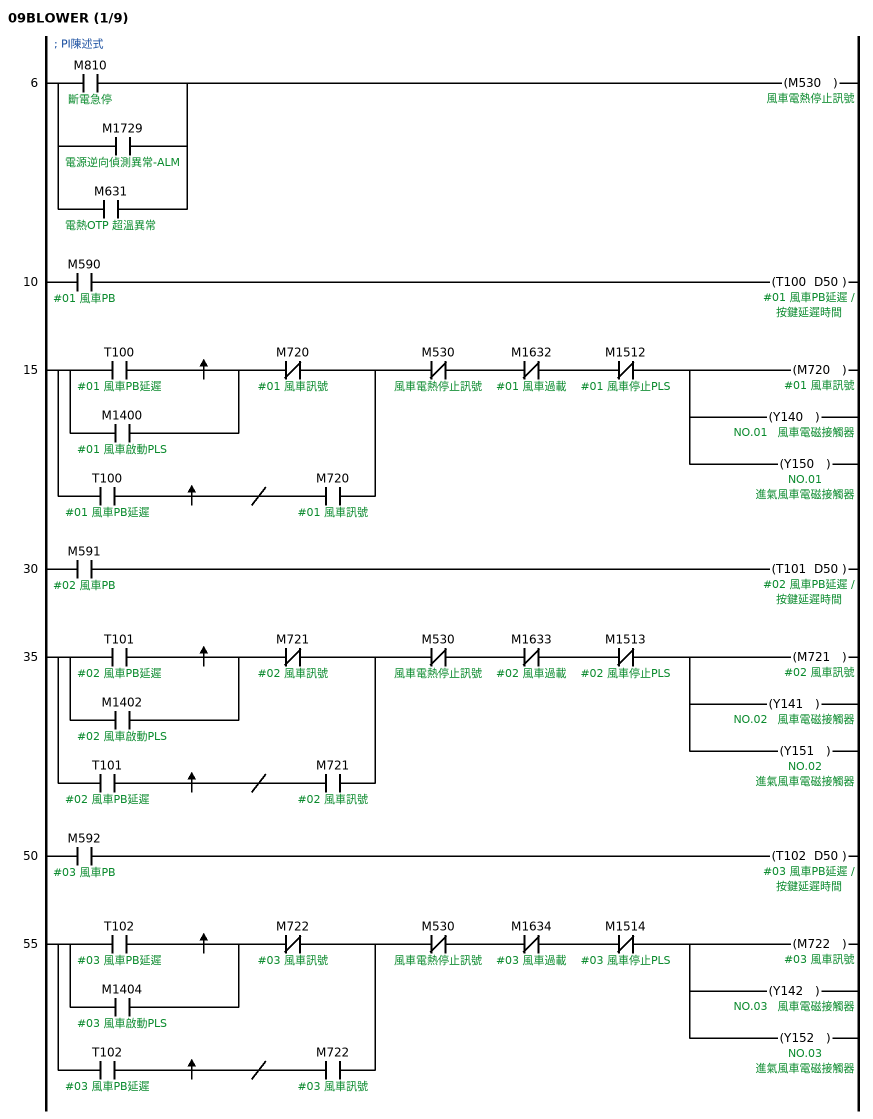
; PI陳述式
6     LD      M810  ; 斷電急停
      OR      M1729  ; 電源逆向偵測異常-ALM
      OR      M631  ; 電熱OTP 超溫異常
      OUT     M530  ; 風車電熱停止訊號
10    LD      M590  ; #01 風車PB
      OUT     T100 D50  ; #01 風車PB延遲 / 按鍵延遲時間
15    LD      T100  ; #01 風車PB延遲
      MEP
      OR      M1400  ; #01 風車啟動PLS
      ANI     M720  ; #01 風車訊號
      LD      T100  ; #01 風車PB延遲
      MEP
      INV
      AND     M720  ; #01 風車訊號
      ORB
      ANI     M530  ; 風車電熱停止訊號
      ANI     M1632  ; #01 風車過載
      ANI     M1512  ; #01 風車停止PLS
      OUT     M720  ; #01 風車訊號
      OUT     Y140  ; NO.01   風車電磁接觸器
      OUT     Y150  ; NO.01   進氣風車電磁接觸器
30    LD      M591  ; #02 風車PB
      OUT     T101 D50  ; #02 風車PB延遲 / 按鍵延遲時間
35    LD      T101  ; #02 風車PB延遲
      MEP
      OR      M1402  ; #02 風車啟動PLS
      ANI     M721  ; #02 風車訊號
      LD      T101  ; #02 風車PB延遲
      MEP
      INV
      AND     M721  ; #02 風車訊號
      ORB
      ANI     M530  ; 風車電熱停止訊號
      ANI     M1633  ; #02 風車過載
      ANI     M1513  ; #02 風車停止PLS
      OUT     M721  ; #02 風車訊號
      OUT     Y141  ; NO.02   風車電磁接觸器
      OUT     Y151  ; NO.02   進氣風車電磁接觸器
50    LD      M592  ; #03 風車PB
      OUT     T102 D50  ; #03 風車PB延遲 / 按鍵延遲時間
55    LD      T102  ; #03 風車PB延遲
      MEP
      OR      M1404  ; #03 風車啟動PLS
      ANI     M722  ; #03 風車訊號
      LD      T102  ; #03 風車PB延遲
      MEP
      INV
      AND     M722  ; #03 風車訊號
      ORB
      ANI     M530  ; 風車電熱停止訊號
      ANI     M1634  ; #03 風車過載
      ANI     M1514  ; #03 風車停止PLS
      OUT     M722  ; #03 風車訊號
      OUT     Y142  ; NO.03   風車電磁接觸器
      OUT     Y152  ; NO.03   進氣風車電磁接觸器
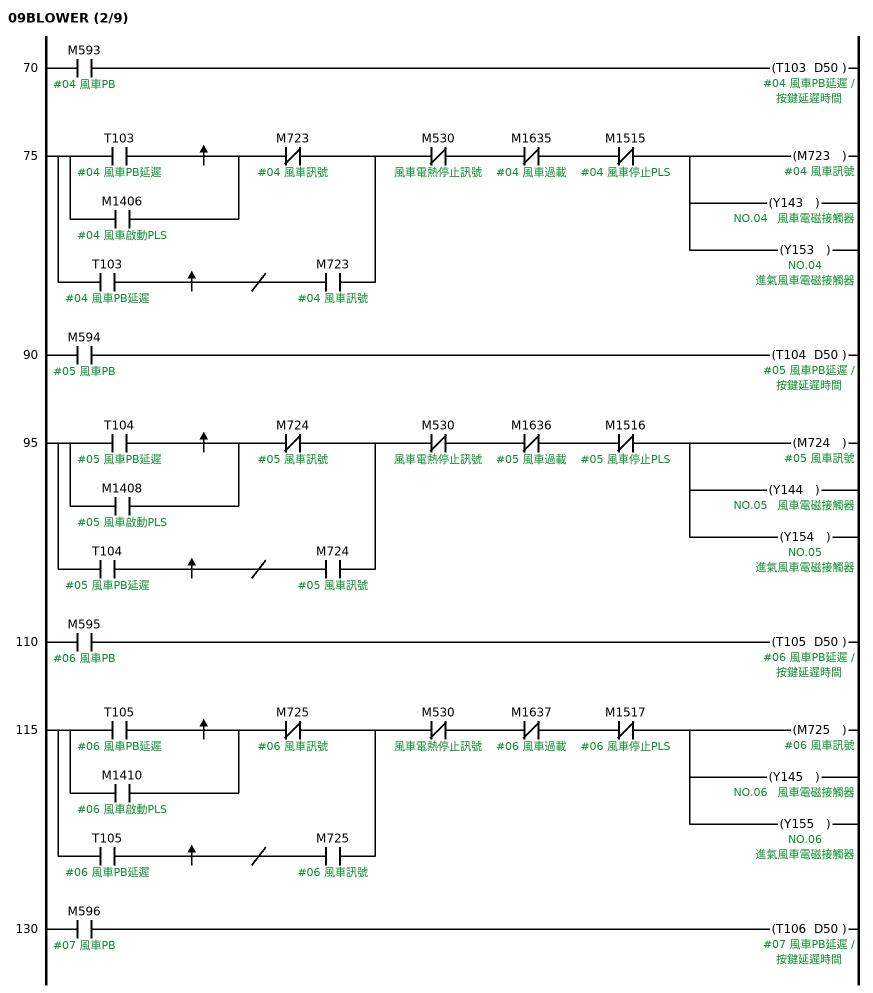
70    LD      M593  ; #04 風車PB
      OUT     T103 D50  ; #04 風車PB延遲 / 按鍵延遲時間
75    LD      T103  ; #04 風車PB延遲
      MEP
      OR      M1406  ; #04 風車啟動PLS
      ANI     M723  ; #04 風車訊號
      LD      T103  ; #04 風車PB延遲
      MEP
      INV
      AND     M723  ; #04 風車訊號
      ORB
      ANI     M530  ; 風車電熱停止訊號
      ANI     M1635  ; #04 風車過載
      ANI     M1515  ; #04 風車停止PLS
      OUT     M723  ; #04 風車訊號
      OUT     Y143  ; NO.04   風車電磁接觸器
      OUT     Y153  ; NO.04   進氣風車電磁接觸器
90    LD      M594  ; #05 風車PB
      OUT     T104 D50  ; #05 風車PB延遲 / 按鍵延遲時間
95    LD      T104  ; #05 風車PB延遲
      MEP
      OR      M1408  ; #05 風車啟動PLS
      ANI     M724  ; #05 風車訊號
      LD      T104  ; #05 風車PB延遲
      MEP
      INV
      AND     M724  ; #05 風車訊號
      ORB
      ANI     M530  ; 風車電熱停止訊號
      ANI     M1636  ; #05 風車過載
      ANI     M1516  ; #05 風車停止PLS
      OUT     M724  ; #05 風車訊號
      OUT     Y144  ; NO.05   風車電磁接觸器
      OUT     Y154  ; NO.05   進氣風車電磁接觸器
110   LD      M595  ; #06 風車PB
      OUT     T105 D50  ; #06 風車PB延遲 / 按鍵延遲時間
115   LD      T105  ; #06 風車PB延遲
      MEP
      OR      M1410  ; #06 風車啟動PLS
      ANI     M725  ; #06 風車訊號
      LD      T105  ; #06 風車PB延遲
      MEP
      INV
      AND     M725  ; #06 風車訊號
      ORB
      ANI     M530  ; 風車電熱停止訊號
      ANI     M1637  ; #06 風車過載
      ANI     M1517  ; #06 風車停止PLS
      OUT     M725  ; #06 風車訊號
      OUT     Y145  ; NO.06   風車電磁接觸器
      OUT     Y155  ; NO.06   進氣風車電磁接觸器
130   LD      M596  ; #07 風車PB
      OUT     T106 D50  ; #07 風車PB延遲 / 按鍵延遲時間
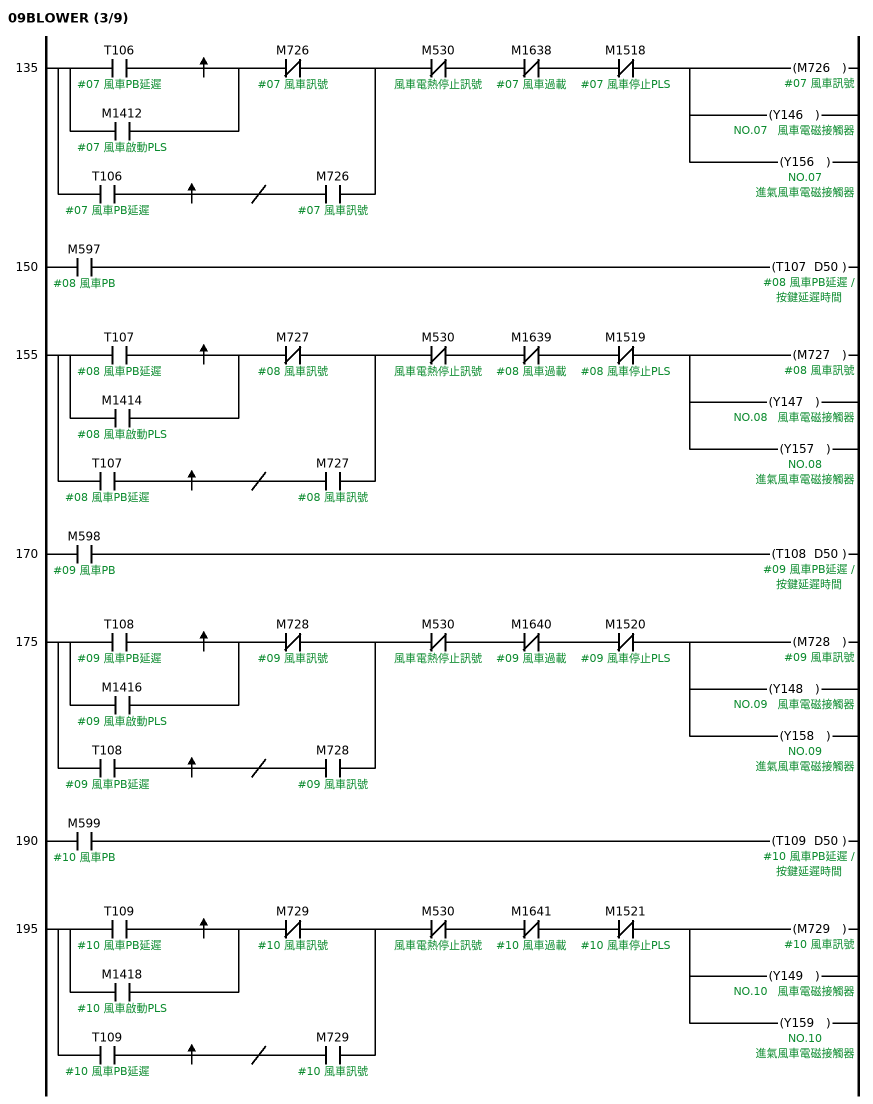
135   LD      T106  ; #07 風車PB延遲
      MEP
      OR      M1412  ; #07 風車啟動PLS
      ANI     M726  ; #07 風車訊號
      LD      T106  ; #07 風車PB延遲
      MEP
      INV
      AND     M726  ; #07 風車訊號
      ORB
      ANI     M530  ; 風車電熱停止訊號
      ANI     M1638  ; #07 風車過載
      ANI     M1518  ; #07 風車停止PLS
      OUT     M726  ; #07 風車訊號
      OUT     Y146  ; NO.07   風車電磁接觸器
      OUT     Y156  ; NO.07   進氣風車電磁接觸器
150   LD      M597  ; #08 風車PB
      OUT     T107 D50  ; #08 風車PB延遲 / 按鍵延遲時間
155   LD      T107  ; #08 風車PB延遲
      MEP
      OR      M1414  ; #08 風車啟動PLS
      ANI     M727  ; #08 風車訊號
      LD      T107  ; #08 風車PB延遲
      MEP
      INV
      AND     M727  ; #08 風車訊號
      ORB
      ANI     M530  ; 風車電熱停止訊號
      ANI     M1639  ; #08 風車過載
      ANI     M1519  ; #08 風車停止PLS
      OUT     M727  ; #08 風車訊號
      OUT     Y147  ; NO.08   風車電磁接觸器
      OUT     Y157  ; NO.08   進氣風車電磁接觸器
170   LD      M598  ; #09 風車PB
      OUT     T108 D50  ; #09 風車PB延遲 / 按鍵延遲時間
175   LD      T108  ; #09 風車PB延遲
      MEP
      OR      M1416  ; #09 風車啟動PLS
      ANI     M728  ; #09 風車訊號
      LD      T108  ; #09 風車PB延遲
      MEP
      INV
      AND     M728  ; #09 風車訊號
      ORB
      ANI     M530  ; 風車電熱停止訊號
      ANI     M1640  ; #09 風車過載
      ANI     M1520  ; #09 風車停止PLS
      OUT     M728  ; #09 風車訊號
      OUT     Y148  ; NO.09   風車電磁接觸器
      OUT     Y158  ; NO.09   進氣風車電磁接觸器
190   LD      M599  ; #10 風車PB
      OUT     T109 D50  ; #10 風車PB延遲 / 按鍵延遲時間
195   LD      T109  ; #10 風車PB延遲
      MEP
      OR      M1418  ; #10 風車啟動PLS
      ANI     M729  ; #10 風車訊號
      LD      T109  ; #10 風車PB延遲
      MEP
      INV
      AND     M729  ; #10 風車訊號
      ORB
      ANI     M530  ; 風車電熱停止訊號
      ANI     M1641  ; #10 風車過載
      ANI     M1521  ; #10 風車停止PLS
      OUT     M729  ; #10 風車訊號
      OUT     Y149  ; NO.10   風車電磁接觸器
      OUT     Y159  ; NO.10   進氣風車電磁接觸器
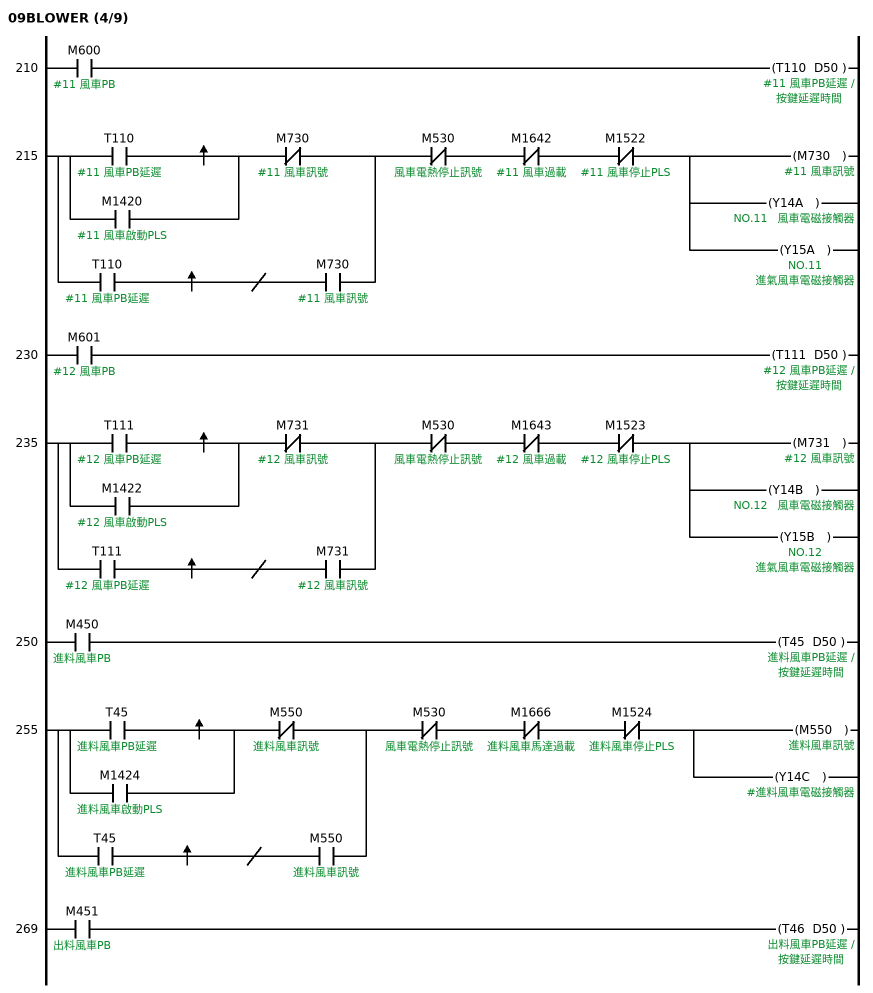
210   LD      M600  ; #11 風車PB
      OUT     T110 D50  ; #11 風車PB延遲 / 按鍵延遲時間
215   LD      T110  ; #11 風車PB延遲
      MEP
      OR      M1420  ; #11 風車啟動PLS
      ANI     M730  ; #11 風車訊號
      LD      T110  ; #11 風車PB延遲
      MEP
      INV
      AND     M730  ; #11 風車訊號
      ORB
      ANI     M530  ; 風車電熱停止訊號
      ANI     M1642  ; #11 風車過載
      ANI     M1522  ; #11 風車停止PLS
      OUT     M730  ; #11 風車訊號
      OUT     Y14A  ; NO.11   風車電磁接觸器
      OUT     Y15A  ; NO.11   進氣風車電磁接觸器
230   LD      M601  ; #12 風車PB
      OUT     T111 D50  ; #12 風車PB延遲 / 按鍵延遲時間
235   LD      T111  ; #12 風車PB延遲
      MEP
      OR      M1422  ; #12 風車啟動PLS
      ANI     M731  ; #12 風車訊號
      LD      T111  ; #12 風車PB延遲
      MEP
      INV
      AND     M731  ; #12 風車訊號
      ORB
      ANI     M530  ; 風車電熱停止訊號
      ANI     M1643  ; #12 風車過載
      ANI     M1523  ; #12 風車停止PLS
      OUT     M731  ; #12 風車訊號
      OUT     Y14B  ; NO.12   風車電磁接觸器
      OUT     Y15B  ; NO.12   進氣風車電磁接觸器
250   LD      M450  ; 進料風車PB
      OUT     T45 D50  ; 進料風車PB延遲 / 按鍵延遲時間
255   LD      T45  ; 進料風車PB延遲
      MEP
      OR      M1424  ; 進料風車啟動PLS
      ANI     M550  ; 進料風車訊號
      LD      T45  ; 進料風車PB延遲
      MEP
      INV
      AND     M550  ; 進料風車訊號
      ORB
      ANI     M530  ; 風車電熱停止訊號
      ANI     M1666  ; 進料風車馬達過載
      ANI     M1524  ; 進料風車停止PLS
      OUT     M550  ; 進料風車訊號
      OUT     Y14C  ; #進料風車電磁接觸器
269   LD      M451  ; 出料風車PB
      OUT     T46 D50  ; 出料風車PB延遲 / 按鍵延遲時間
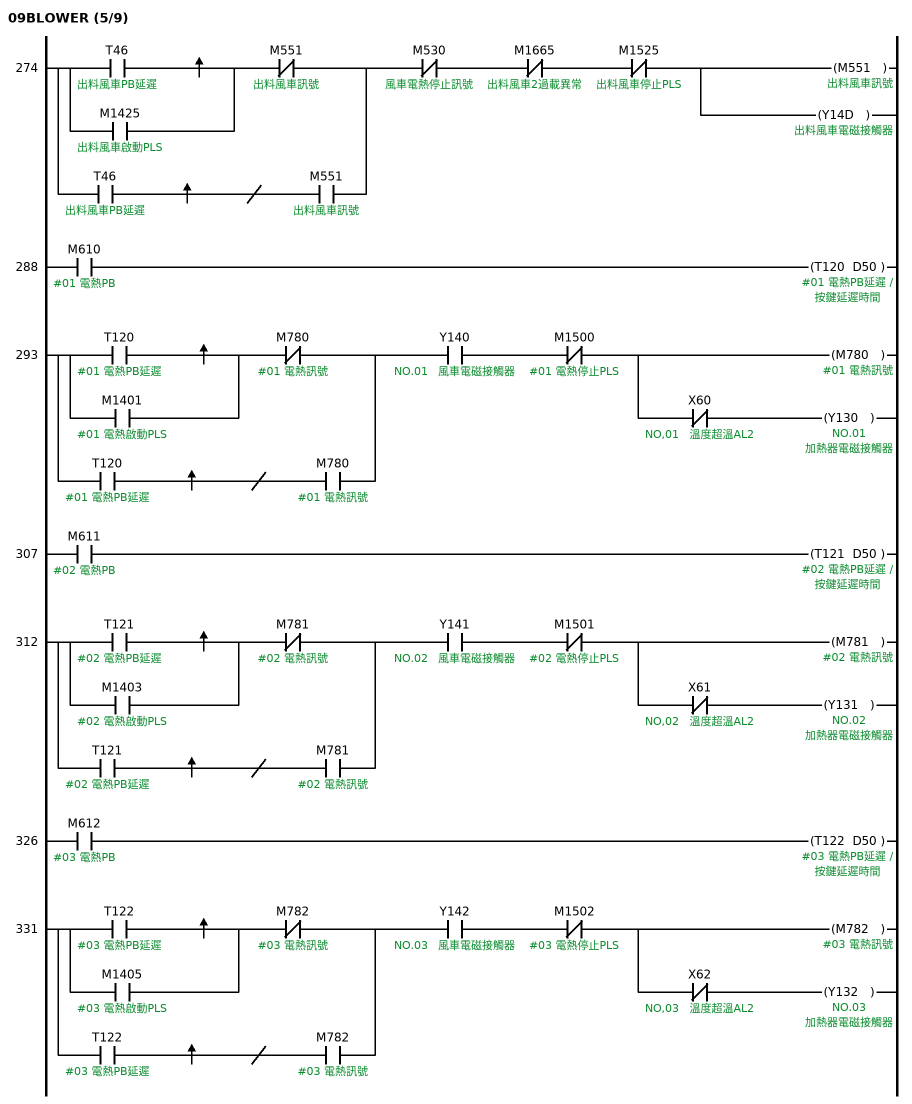
274   LD      T46  ; 出料風車PB延遲
      MEP
      OR      M1425  ; 出料風車啟動PLS
      ANI     M551  ; 出料風車訊號
      LD      T46  ; 出料風車PB延遲
      MEP
      INV
      AND     M551  ; 出料風車訊號
      ORB
      ANI     M530  ; 風車電熱停止訊號
      ANI     M1665  ; 出料風車2過載異常
      ANI     M1525  ; 出料風車停止PLS
      OUT     M551  ; 出料風車訊號
      OUT     Y14D  ; 出料風車電磁接觸器
288   LD      M610  ; #01 電熱PB
      OUT     T120 D50  ; #01 電熱PB延遲 / 按鍵延遲時間
293   LD      T120  ; #01 電熱PB延遲
      MEP
      OR      M1401  ; #01 電熱啟動PLS
      ANI     M780  ; #01 電熱訊號
      LD      T120  ; #01 電熱PB延遲
      MEP
      INV
      AND     M780  ; #01 電熱訊號
      ORB
      AND     Y140  ; NO.01   風車電磁接觸器
      ANI     M1500  ; #01 電熱停止PLS
      OUT     M780  ; #01 電熱訊號
      ANI     X60  ; NO,01   溫度超溫AL2
      OUT     Y130  ; NO.01   加熱器電磁接觸器
307   LD      M611  ; #02 電熱PB
      OUT     T121 D50  ; #02 電熱PB延遲 / 按鍵延遲時間
312   LD      T121  ; #02 電熱PB延遲
      MEP
      OR      M1403  ; #02 電熱啟動PLS
      ANI     M781  ; #02 電熱訊號
      LD      T121  ; #02 電熱PB延遲
      MEP
      INV
      AND     M781  ; #02 電熱訊號
      ORB
      AND     Y141  ; NO.02   風車電磁接觸器
      ANI     M1501  ; #02 電熱停止PLS
      OUT     M781  ; #02 電熱訊號
      ANI     X61  ; NO,02   溫度超溫AL2
      OUT     Y131  ; NO.02   加熱器電磁接觸器
326   LD      M612  ; #03 電熱PB
      OUT     T122 D50  ; #03 電熱PB延遲 / 按鍵延遲時間
331   LD      T122  ; #03 電熱PB延遲
      MEP
      OR      M1405  ; #03 電熱啟動PLS
      ANI     M782  ; #03 電熱訊號
      LD      T122  ; #03 電熱PB延遲
      MEP
      INV
      AND     M782  ; #03 電熱訊號
      ORB
      AND     Y142  ; NO.03   風車電磁接觸器
      ANI     M1502  ; #03 電熱停止PLS
      OUT     M782  ; #03 電熱訊號
      ANI     X62  ; NO,03   溫度超溫AL2
      OUT     Y132  ; NO.03   加熱器電磁接觸器
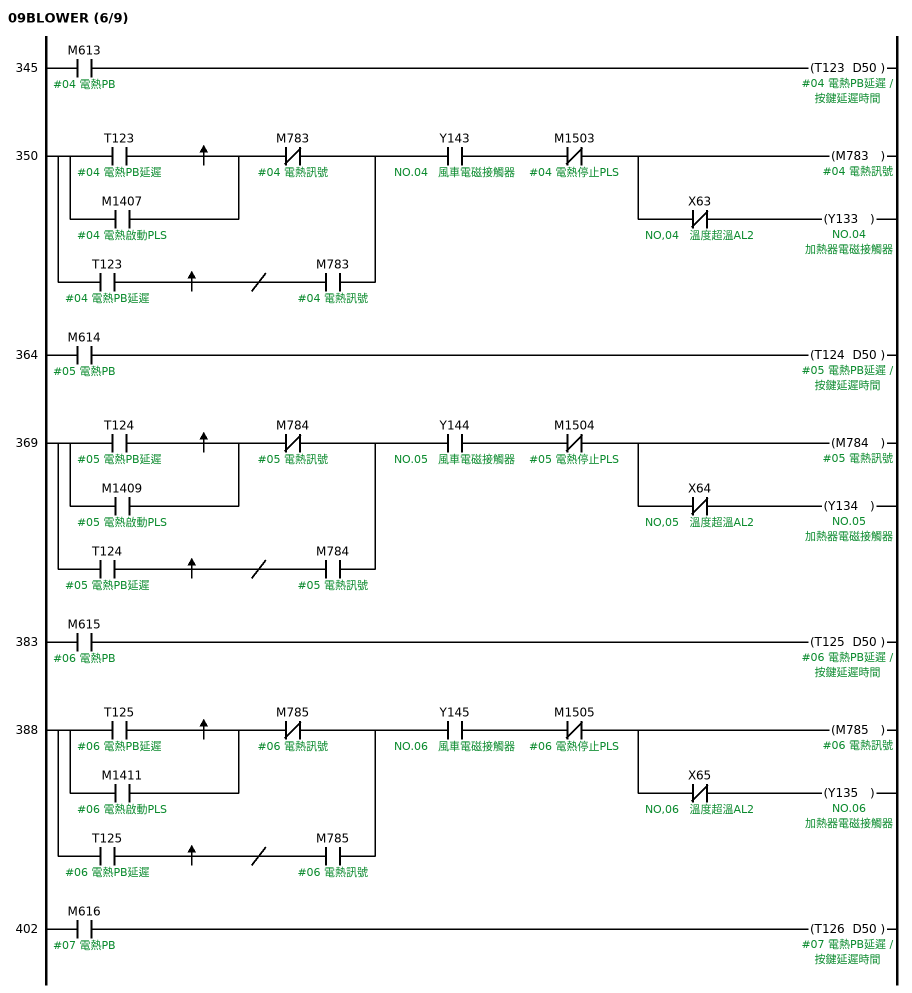
345   LD      M613  ; #04 電熱PB
      OUT     T123 D50  ; #04 電熱PB延遲 / 按鍵延遲時間
350   LD      T123  ; #04 電熱PB延遲
      MEP
      OR      M1407  ; #04 電熱啟動PLS
      ANI     M783  ; #04 電熱訊號
      LD      T123  ; #04 電熱PB延遲
      MEP
      INV
      AND     M783  ; #04 電熱訊號
      ORB
      AND     Y143  ; NO.04   風車電磁接觸器
      ANI     M1503  ; #04 電熱停止PLS
      OUT     M783  ; #04 電熱訊號
      ANI     X63  ; NO,04   溫度超溫AL2
      OUT     Y133  ; NO.04   加熱器電磁接觸器
364   LD      M614  ; #05 電熱PB
      OUT     T124 D50  ; #05 電熱PB延遲 / 按鍵延遲時間
369   LD      T124  ; #05 電熱PB延遲
      MEP
      OR      M1409  ; #05 電熱啟動PLS
      ANI     M784  ; #05 電熱訊號
      LD      T124  ; #05 電熱PB延遲
      MEP
      INV
      AND     M784  ; #05 電熱訊號
      ORB
      AND     Y144  ; NO.05   風車電磁接觸器
      ANI     M1504  ; #05 電熱停止PLS
      OUT     M784  ; #05 電熱訊號
      ANI     X64  ; NO,05   溫度超溫AL2
      OUT     Y134  ; NO.05   加熱器電磁接觸器
383   LD      M615  ; #06 電熱PB
      OUT     T125 D50  ; #06 電熱PB延遲 / 按鍵延遲時間
388   LD      T125  ; #06 電熱PB延遲
      MEP
      OR      M1411  ; #06 電熱啟動PLS
      ANI     M785  ; #06 電熱訊號
      LD      T125  ; #06 電熱PB延遲
      MEP
      INV
      AND     M785  ; #06 電熱訊號
      ORB
      AND     Y145  ; NO.06   風車電磁接觸器
      ANI     M1505  ; #06 電熱停止PLS
      OUT     M785  ; #06 電熱訊號
      ANI     X65  ; NO,06   溫度超溫AL2
      OUT     Y135  ; NO.06   加熱器電磁接觸器
402   LD      M616  ; #07 電熱PB
      OUT     T126 D50  ; #07 電熱PB延遲 / 按鍵延遲時間
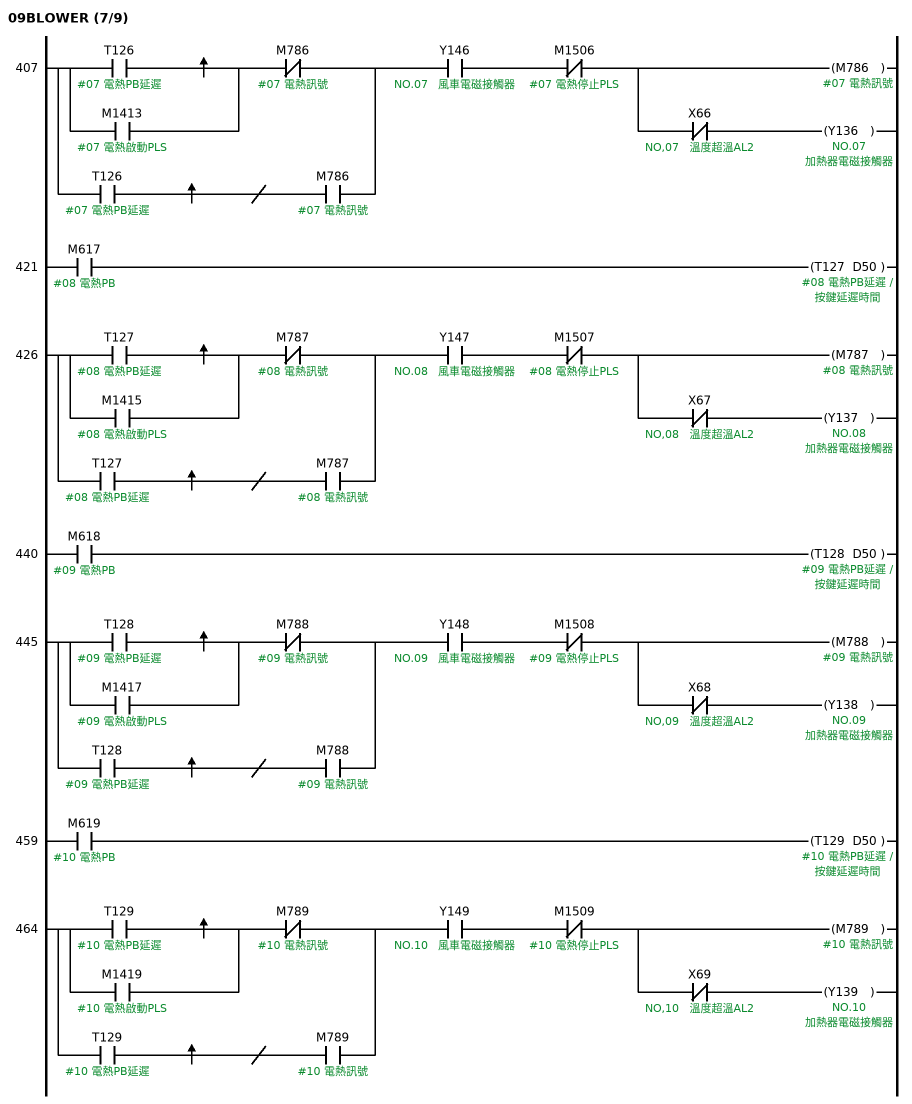
407   LD      T126  ; #07 電熱PB延遲
      MEP
      OR      M1413  ; #07 電熱啟動PLS
      ANI     M786  ; #07 電熱訊號
      LD      T126  ; #07 電熱PB延遲
      MEP
      INV
      AND     M786  ; #07 電熱訊號
      ORB
      AND     Y146  ; NO.07   風車電磁接觸器
      ANI     M1506  ; #07 電熱停止PLS
      OUT     M786  ; #07 電熱訊號
      ANI     X66  ; NO,07   溫度超溫AL2
      OUT     Y136  ; NO.07   加熱器電磁接觸器
421   LD      M617  ; #08 電熱PB
      OUT     T127 D50  ; #08 電熱PB延遲 / 按鍵延遲時間
426   LD      T127  ; #08 電熱PB延遲
      MEP
      OR      M1415  ; #08 電熱啟動PLS
      ANI     M787  ; #08 電熱訊號
      LD      T127  ; #08 電熱PB延遲
      MEP
      INV
      AND     M787  ; #08 電熱訊號
      ORB
      AND     Y147  ; NO.08   風車電磁接觸器
      ANI     M1507  ; #08 電熱停止PLS
      OUT     M787  ; #08 電熱訊號
      ANI     X67  ; NO,08   溫度超溫AL2
      OUT     Y137  ; NO.08   加熱器電磁接觸器
440   LD      M618  ; #09 電熱PB
      OUT     T128 D50  ; #09 電熱PB延遲 / 按鍵延遲時間
445   LD      T128  ; #09 電熱PB延遲
      MEP
      OR      M1417  ; #09 電熱啟動PLS
      ANI     M788  ; #09 電熱訊號
      LD      T128  ; #09 電熱PB延遲
      MEP
      INV
      AND     M788  ; #09 電熱訊號
      ORB
      AND     Y148  ; NO.09   風車電磁接觸器
      ANI     M1508  ; #09 電熱停止PLS
      OUT     M788  ; #09 電熱訊號
      ANI     X68  ; NO,09   溫度超溫AL2
      OUT     Y138  ; NO.09   加熱器電磁接觸器
459   LD      M619  ; #10 電熱PB
      OUT     T129 D50  ; #10 電熱PB延遲 / 按鍵延遲時間
464   LD      T129  ; #10 電熱PB延遲
      MEP
      OR      M1419  ; #10 電熱啟動PLS
      ANI     M789  ; #10 電熱訊號
      LD      T129  ; #10 電熱PB延遲
      MEP
      INV
      AND     M789  ; #10 電熱訊號
      ORB
      AND     Y149  ; NO.10   風車電磁接觸器
      ANI     M1509  ; #10 電熱停止PLS
      OUT     M789  ; #10 電熱訊號
      ANI     X69  ; NO,10   溫度超溫AL2
      OUT     Y139  ; NO.10   加熱器電磁接觸器
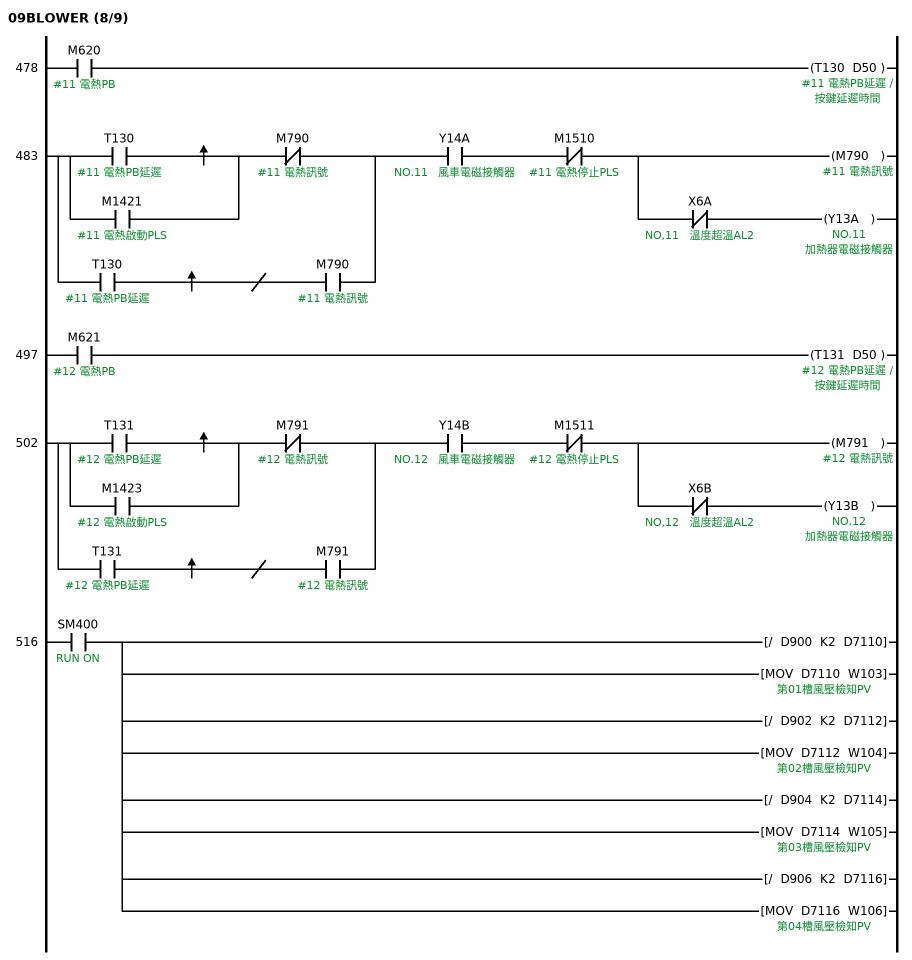
478   LD      M620  ; #11 電熱PB
      OUT     T130 D50  ; #11 電熱PB延遲 / 按鍵延遲時間
483   LD      T130  ; #11 電熱PB延遲
      MEP
      OR      M1421  ; #11 電熱啟動PLS
      ANI     M790  ; #11 電熱訊號
      LD      T130  ; #11 電熱PB延遲
      MEP
      INV
      AND     M790  ; #11 電熱訊號
      ORB
      AND     Y14A  ; NO.11   風車電磁接觸器
      ANI     M1510  ; #11 電熱停止PLS
      OUT     M790  ; #11 電熱訊號
      ANI     X6A  ; NO,11   溫度超溫AL2
      OUT     Y13A  ; NO.11   加熱器電磁接觸器
497   LD      M621  ; #12 電熱PB
      OUT     T131 D50  ; #12 電熱PB延遲 / 按鍵延遲時間
502   LD      T131  ; #12 電熱PB延遲
      MEP
      OR      M1423  ; #12 電熱啟動PLS
      ANI     M791  ; #12 電熱訊號
      LD      T131  ; #12 電熱PB延遲
      MEP
      INV
      AND     M791  ; #12 電熱訊號
      ORB
      AND     Y14B  ; NO.12   風車電磁接觸器
      ANI     M1511  ; #12 電熱停止PLS
      OUT     M791  ; #12 電熱訊號
      ANI     X6B  ; NO,12   溫度超溫AL2
      OUT     Y13B  ; NO.12   加熱器電磁接觸器
516   LD      SM400  ; RUN ON
      /       D900 K2 D7110
      MOV     D7110 W103  ; 第01槽風壓檢知PV
      /       D902 K2 D7112
      MOV     D7112 W104  ; 第02槽風壓檢知PV
      /       D904 K2 D7114
      MOV     D7114 W105  ; 第03槽風壓檢知PV
      /       D906 K2 D7116
      MOV     D7116 W106  ; 第04槽風壓檢知PV
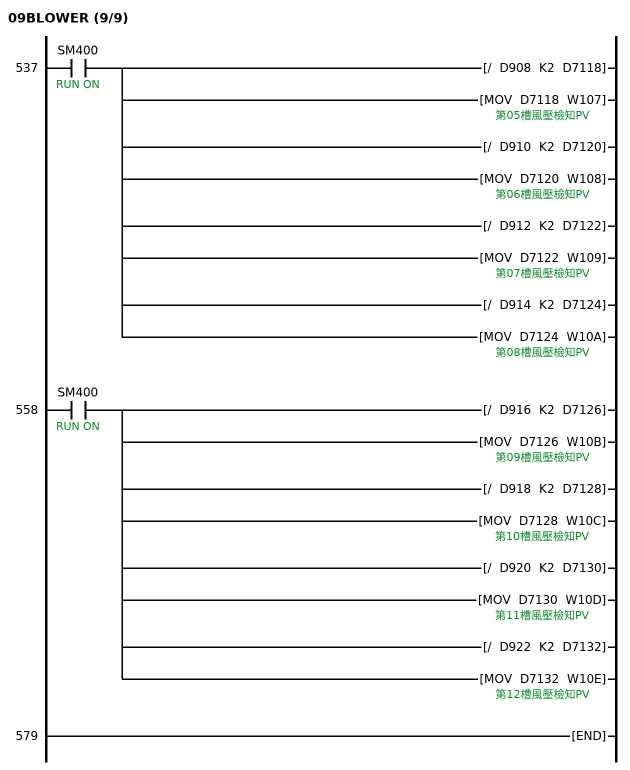
537   LD      SM400  ; RUN ON
      /       D908 K2 D7118
      MOV     D7118 W107  ; 第05槽風壓檢知PV
      /       D910 K2 D7120
      MOV     D7120 W108  ; 第06槽風壓檢知PV
      /       D912 K2 D7122
      MOV     D7122 W109  ; 第07槽風壓檢知PV
      /       D914 K2 D7124
      MOV     D7124 W10A  ; 第08槽風壓檢知PV
558   LD      SM400  ; RUN ON
      /       D916 K2 D7126
      MOV     D7126 W10B  ; 第09槽風壓檢知PV
      /       D918 K2 D7128
      MOV     D7128 W10C  ; 第10槽風壓檢知PV
      /       D920 K2 D7130
      MOV     D7130 W10D  ; 第11槽風壓檢知PV
      /       D922 K2 D7132
      MOV     D7132 W10E  ; 第12槽風壓檢知PV
579   END
END_PROGRAM

PROGRAM 10YIELD
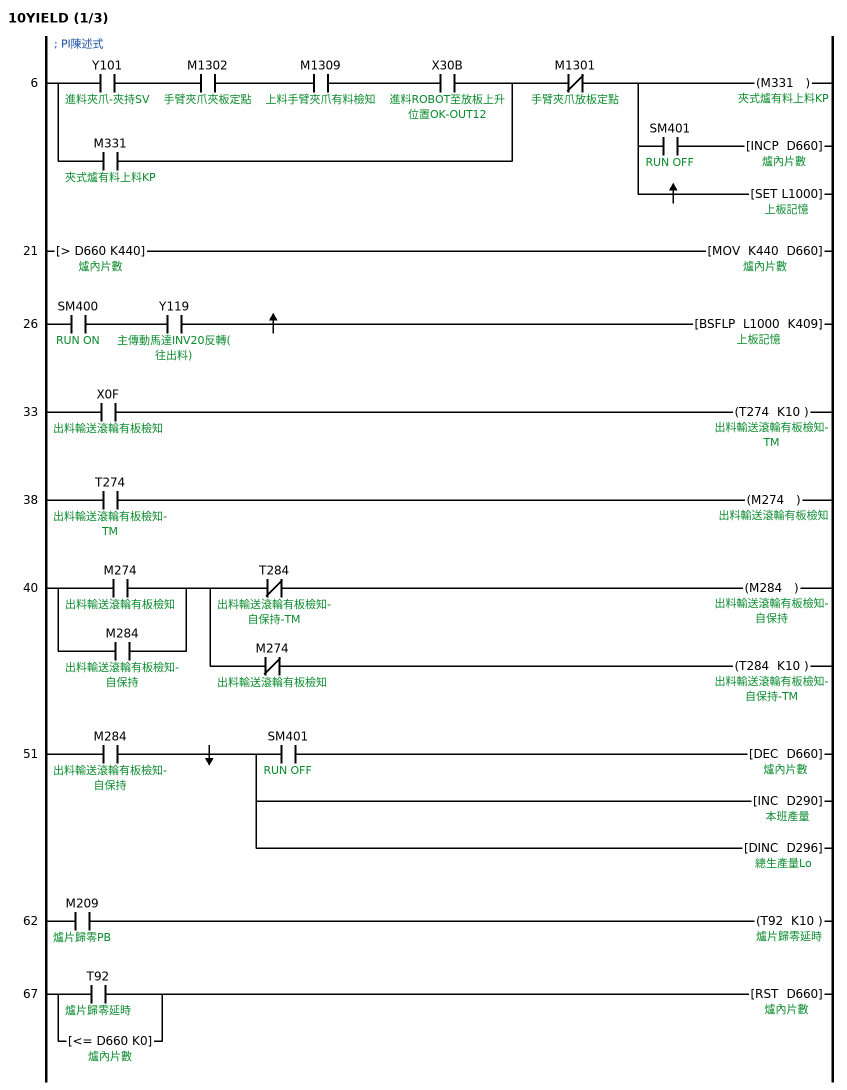
; PI陳述式
6     LD      Y101  ; 進料夾爪-夾持SV
      AND     M1302  ; 手臂夾爪夾板定點
      AND     M1309  ; 上料手臂夾爪有料檢知
      AND     X30B  ; 進料ROBOT至放板上升位置OK-OUT12
      OR      M331  ; 夾式爐有料上料KP
      ANI     M1301  ; 手臂夾爪放板定點
      OUT     M331  ; 夾式爐有料上料KP
      MPS
      AND     SM401  ; RUN OFF
      INCP    D660  ; 爐內片數
      MPP
      MEP
      SET     L1000  ; 上板記憶
21    LD>     D660 K440  ; 爐內片數
      MOV     K440 D660
26    LD      SM400  ; RUN ON
      AND     Y119  ; 主傳動馬達INV20反轉(往出料)
      MEP
      BSFLP   L1000 K409
33    LD      X0F  ; 出料輸送滾輪有板檢知
      OUT     T274 K10  ; 出料輸送滾輪有板檢知-TM
38    LD      T274  ; 出料輸送滾輪有板檢知-TM
      OUT     M274  ; 出料輸送滾輪有板檢知
40    LD      M274  ; 出料輸送滾輪有板檢知
      OR      M284  ; 出料輸送滾輪有板檢知-自保持
      MPS
      ANI     T284  ; 出料輸送滾輪有板檢知-自保持-TM
      OUT     M284  ; 出料輸送滾輪有板檢知-自保持
      MPP
      ANI     M274  ; 出料輸送滾輪有板檢知
      OUT     T284 K10  ; 出料輸送滾輪有板檢知-自保持-TM
51    LD      M284  ; 出料輸送滾輪有板檢知-自保持
      MEF
      MPS
      AND     SM401  ; RUN OFF
      DEC     D660
      MPP
      INC     D290  ; 本班產量
      DINC    D296  ; 總生產量Lo
62    LD      M209  ; 爐片歸零PB
      OUT     T92 K10  ; 爐片歸零延時
67    LD      T92  ; 爐片歸零延時
      OR<=    D660 K0  ; 爐內片數
      RST     D660  ; 爐內片數
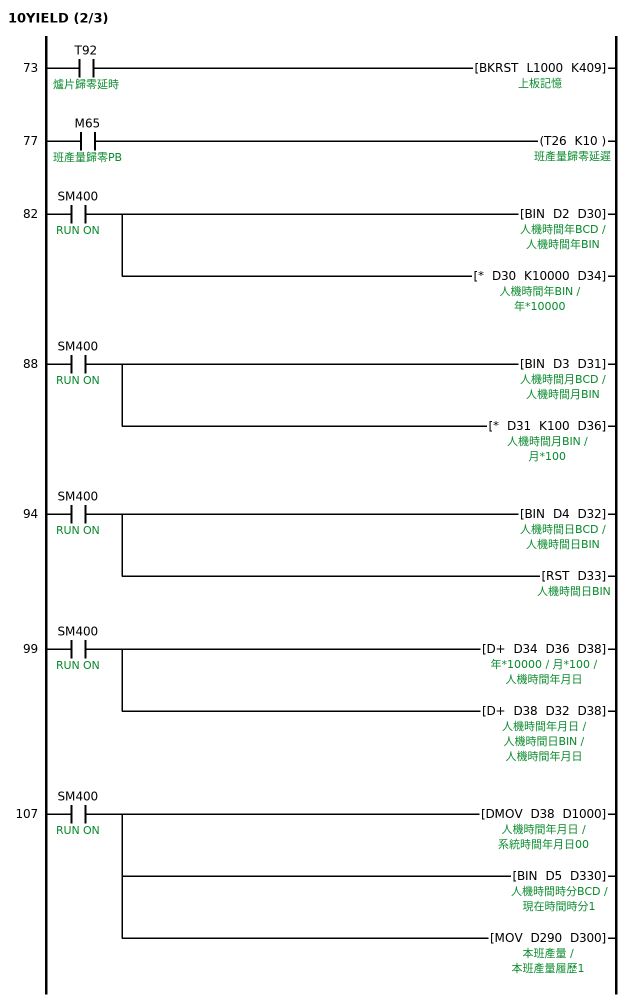
73    LD      T92  ; 爐片歸零延時
      BKRST   L1000 K409
77    LD      M65  ; 班產量歸零PB
      OUT     T26 K10  ; 班產量歸零延遲
82    LD      SM400  ; RUN ON
      BIN     D2 D30  ; 人機時間年BCD / 人機時間年BIN
      *       D30 K10000 D34  ; 年*10000
88    LD      SM400  ; RUN ON
      BIN     D3 D31  ; 人機時間月BCD / 人機時間月BIN
      *       D31 K100 D36  ; 月*100
94    LD      SM400  ; RUN ON
      BIN     D4 D32  ; 人機時間日BCD / 人機時間日BIN
      RST     D33  ; 人機時間日BIN
99    LD      SM400  ; RUN ON
      D+      D34 D36 D38  ; 人機時間年月日
      D+      D38 D32 D38
107   LD      SM400  ; RUN ON
      DMOV    D38 D1000  ; 系統時間年月日00
      BIN     D5 D330  ; 人機時間時分BCD / 現在時間時分1
      MOV     D290 D300  ; 本班產量履歷1
